  // ------------------------------------------
  // SyncMode : SERVER_TO_CLIENT 
  // ------------------------------------------
  12 : // Conflict triggerd by PLC ?  
       IF ( NOT AxesGroup.State.SyncStatePlc.InSync.Frame )
       THEN
         // search for changed index  
         FOR _rSyncIdx := 0 TO AxesGroup.State.UnifiedFrameIndex
         DO
           IF ( AxesGroup.State.DataChanged.Frame[_rSyncIdx] )
           THEN
             // set timeout
             SetTimeout(PT := _rTimeout, rTimer := _rTimer);
             // inc step counter
            _rStep := 20; // -> read RC data and write it to PLC                  
             EXIT;
					 END_IF
         END_FOR

         // Create log entry
         CreateLogMessagePara3 ( Timestamp   := SystemTime,
                                 MessageType := MessageType.CMD,
                                 Severity    := Severity.DEBUG,
                                 MessageCode := 0,
                                 MessageText := 'SyncFrameData: Synchronization of Frame[{1}] triggered by PLC, SyncMode = {2}, SyncTime = {3}, SyncDirection = RC -> PLC',
                                 Para1       :=  DINT_TO_STRING(_rSyncIdx),
                                 Para2       :=  SYNC_MODE_TO_STRING(AxesGroup.Parameter.Plc.Parameter.SynchronizationModes.Frame[SyncTime.AFTER_START_UP]),
                                 Para3       :=  SYNC_TIME_TO_STRING(SyncTime.AFTER_START_UP));
                                 RETURN;
       END_IF
   
       // Conflict triggered by RC ?
       IF ( NOT AxesGroup.State.SyncStateRc.InSync.Frame )
       THEN
         // get changed index 
        _rSyncIdx := LIMIT(0, AxesGroup.State.SyncStateRc.UnSyncNo.Frame, AxesGroup.State.UnifiedFrameIndex);
         // set timeout
         SetTimeout(PT := _rTimeout, rTimer := _rTimer);
         // inc step counter
        _rStep := 20; // -> read RC data and write it to PLC

         // Create log entry
         CreateLogMessagePara3 ( Timestamp   := SystemTime,
                                 MessageType := MessageType.CMD,
                                 Severity    := Severity.DEBUG,
                                 MessageCode := 0,
                                 MessageText := 'SyncFrameData: Synchronization of Frame[{1}] triggered by RC, SyncMode = {2}, SyncTime = {3}, SyncDirection = RC -> PLC',
                                 Para1       :=  DINT_TO_STRING(_rSyncIdx),
                                 Para2       :=  SYNC_MODE_TO_STRING(AxesGroup.Parameter.Plc.Parameter.SynchronizationModes.Frame[SyncTime.AFTER_START_UP]),
                                 Para3       :=  SYNC_TIME_TO_STRING(SyncTime.AFTER_START_UP));
                                 RETURN;
			 END_IF
       
       // set timeout
       SetTimeout(PT := _rTimeout, rTimer := _rTimer);
       // jump back
      _rStep := 10;
  

  // ------------------------------------------
  // SyncMode : AUTOMATIC 
  // ------------------------------------------
  13 : // Conflict triggerd by PLC ?  
       IF ( NOT AxesGroup.State.SyncStatePlc.InSync.Frame )
       THEN
         // search for changed index  
         FOR _rSyncIdx := 0 TO AxesGroup.State.UnifiedFrameIndex
         DO
           IF ( AxesGroup.State.DataChanged.Frame[_rSyncIdx] )
           THEN
             // set timeout
             SetTimeout(PT := _rTimeout, rTimer := _rTimer);
             // inc step counter
            _rStep := 30; // -> write PLC data to RC                  
             EXIT;
					 END_IF
         END_FOR
         
         // Create log entry
         CreateLogMessagePara3 ( Timestamp   := SystemTime,
                                 MessageType := MessageType.CMD,
                                 Severity    := Severity.DEBUG,
                                 MessageCode := 0,
                                 MessageText := 'SyncFrameData: Synchronization of Frame[{1}] triggered by PLC, SyncMode = {2}, SyncTime = {3}, SyncDirection = PLC -> RC',
                                 Para1       :=  DINT_TO_STRING(_rSyncIdx),
                                 Para2       :=  SYNC_MODE_TO_STRING(AxesGroup.Parameter.Plc.Parameter.SynchronizationModes.Frame[SyncTime.AFTER_START_UP]),
                                 Para3       :=  SYNC_TIME_TO_STRING(SyncTime.AFTER_START_UP));
                                 RETURN;
       END_IF
   
       // Conflict triggered by RC ?
       IF ( NOT AxesGroup.State.SyncStateRc.InSync.Frame )
       THEN
         // get changed index 
        _rSyncIdx := LIMIT(0, AxesGroup.State.SyncStateRc.UnSyncNo.Frame, AxesGroup.State.UnifiedFrameIndex);
         // set timeout
         SetTimeout(PT := _rTimeout, rTimer := _rTimer);
         // inc step counter
        _rStep := 20; // -> read RC data an write it to PLC

         // Create log entry
         CreateLogMessagePara3 ( Timestamp   := SystemTime,
                                 MessageType := MessageType.CMD,
                                 Severity    := Severity.DEBUG,
                                 MessageCode := 0,
                                 MessageText := 'SyncFrameData: Synchronization of Frame[{1}] triggered by RC, SyncMode = {2}, SyncTime = {3}, SyncDirection = RC -> PLC',
                                 Para1       :=  DINT_TO_STRING(_rSyncIdx),
                                 Para2       :=  SYNC_MODE_TO_STRING(AxesGroup.Parameter.Plc.Parameter.SynchronizationModes.Frame[SyncTime.AFTER_START_UP]),
                                 Para3       :=  SYNC_TIME_TO_STRING(SyncTime.AFTER_START_UP));
                                 RETURN;
			 END_IF
       
       // set timeout
       SetTimeout(PT := _rTimeout, rTimer := _rTimer);
       // jump back
      //_rStep := 10;


  // ------------------------------------------
  // Read Data from RC and write it to PLC
  // ------------------------------------------
  20 : IF (( NOT _readFrameData.Busy  ) AND 
           ( NOT _readFrameData.Error ))
       THEN
         // set command parameter
        _readFrameData.ParCmd.FrameNo := _rSyncIdx;      
         // execute command
        _readFrameData.Execute := TRUE;
         // set timeout
         SetTimeout(PT := _rTimeout, rTimer := _rTimer);
         // inc step counter
        _rStep := _rStep + 1;
       ELSE
         // check error ? 
         IF (_readFrameData.Error)
         THEN
           ErrorID     := _readFrameData.ErrorID;
           ErrorAddTxt := _readFrameData.ErrorAddTxt;
         END_IF  
       
         // timeout exceeded ? 
         IF (CheckTimeout(_rTimer) = RobotLibraryConstants.OK)
         THEN
           ErrorAddTxt := CONCAT(_stepName, DINT_TO_STRING(_rStep));
           SetError( ErrorID := RobotLibraryErrorIdEnum.ERR_TIMEOUT_CMD, Overwrite := FALSE);
         END_IF
       END_IF
 
  21 : IF (( NOT _readFrameData.Busy  ) AND
           ( NOT _readFrameData.Error ) AND
           (     _readFrameData.Done  ))
       THEN
         // reset execution
        _readFrameData.Execute := FALSE;
         // update internal frame data
         FrameData[_rSyncIdx].Data := _readFrameData.OutCmd.FrameData;         
        _frameData[_rSyncIdx].Data := _readFrameData.OutCmd.FrameData;
         // set available bit
         FrameData[_rSyncIdx].Available := TRUE;
        _frameData[_rSyncIdx].Available := TRUE;
         // set timeout
         SetTimeout(PT := _rTimeout, rTimer := _rTimer);
         // inc step counter
        _rStep := 10; // -> jump to after startup           
       ELSE
         // check error ? 
         IF (_readFrameData.Error)
         THEN
           ErrorID     := _readFrameData.ErrorID;
           ErrorAddTxt := _readFrameData.ErrorAddTxt;           
           // reset available bit
           FrameData[_rSyncIdx].Available := FALSE;
          _frameData[_rSyncIdx].Available := FALSE;
         END_IF  
       
         // timeout exceeded ? 
         IF (CheckTimeout(_rTimer) = RobotLibraryConstants.OK)
         THEN
           ErrorAddTxt := CONCAT(_stepName, DINT_TO_STRING(_rStep));
           SetError( ErrorID := RobotLibraryErrorIdEnum.ERR_TIMEOUT_CMD, Overwrite := FALSE);
         END_IF
       END_IF


  // ------------------------------------------
  // Write data from PLC to RC
  // ------------------------------------------
  30 : IF (( NOT _writeFrameData.Busy  ) AND 
           ( NOT _writeFrameData.Error ))
       THEN
         // set command parameter
        _writeFrameData.ParCmd.FrameNo   := _rSyncIdx;      
        _writeFrameData.ParCmd.FrameData :=  FrameData[_rSyncIdx].Data;
         // execute command
        _writeFrameData.Execute := TRUE;
         // set timeout
         SetTimeout(PT := _rTimeout, rTimer := _rTimer);
         // inc step counter
        _rStep := _rStep + 1;
       ELSE
         // check error ? 
         IF (_writeFrameData.Error)
         THEN
           ErrorID     := _writeFrameData.ErrorID;
           ErrorAddTxt := _writeFrameData.ErrorAddTxt;;
         END_IF  
       
         // timeout exceeded ? 
         IF (CheckTimeout(_rTimer) = RobotLibraryConstants.OK)
         THEN
           ErrorAddTxt := CONCAT(_stepName, DINT_TO_STRING(_rStep));
           SetError( ErrorID := RobotLibraryErrorIdEnum.ERR_TIMEOUT_CMD, Overwrite := FALSE);
         END_IF
       END_IF
 
  31 : IF (( NOT _writeFrameData.Busy  ) AND
           ( NOT _writeFrameData.Error ) AND
           (     _writeFrameData.Done  ))
       THEN
         // execute command
        _writeFrameData.Execute := FALSE;      
         // update internal frame data
        _frameData[_rSyncIdx] := FrameData[_rSyncIdx]; 
         // set available bit
         FrameData[_rSyncIdx].Available := TRUE; 
        _frameData[_rSyncIdx].Available := TRUE;         
         // set timeout
         SetTimeout(PT := _rTimeout, rTimer := _rTimer);
         // inc step counter
        _rStep := 10; // -> jump to after startup;           
       ELSE
         // check error ? 
         IF (_writeFrameData.Error)
         THEN
           SetWarning( WarningID := RobotLibraryWarningIdEnum.WARN_FRAME_SYNC_FAILED_BY_ERROR_OF_READ_OR_WRITE_CMD, Overwrite := TRUE);    
           // reset available bit
           FrameData[_rSyncIdx].Available := FALSE;
          _frameData[_rSyncIdx].Available := FALSE;
         END_IF  
       
         // timeout exceeded ? 
         IF (CheckTimeout(_rTimer) = RobotLibraryConstants.OK)
         THEN
           ErrorAddTxt := CONCAT(_stepName, DINT_TO_STRING(_rStep));
           SetError( ErrorID := RobotLibraryErrorIdEnum.ERR_TIMEOUT_CMD, Overwrite := FALSE);
         END_IF
       END_IF
       
ELSE
  // invalid step
  ErrorID     := RobotLibraryErrorIdEnum.ERR_INVALID_STEP;
  ErrorAddTxt := CONCAT(_stepName , DINT_TO_STRING(_stepCmd));
END_CASE  
                
END_METHOD

METHOD PRIVATE HandleSyncLoadData
VAR_IN_OUT
   /// Robot assignment of function
  AxesGroup : AxesGroup;
  /// LoadData stored on PLC.For more information refer to 5.5.6.4
  LoadData  : ARRAY[*] OF Load;
END_VAR 

VAR
  /// Internal step counter name
 _stepName        : STRING;    
  /// Internal reference to step counter
 _rStep           : REFERENCE TO DINT;
  /// Internal reference to timer
 _rTimer          : REFERENCE TO TON;
  /// Internal reference to timeout
 _rTimeout        : REFERENCE TO TIME; 
  /// Internal reference to synchroniztion index
 _rSyncIdx        : REFERENCE TO USINT;
  /// internal bit for condition found
 _found           : BOOL;
  /// empty data set to reset all DataChanged bits
 _dataChangedNone : AxesGroupStateDataChanged;
  /// internal index for loops
 _idx             : DINT;
  /// internal Start index for loops
 _idxStart        : USINT;
END_VAR
                  // Set internal references 
_stepName      :=   '_stepSyncLoadData = ';
_rStep       REF=    _stepSyncLoadData;
_rTimer      REF=   _timerSyncLoadData;
_rTimeout    REF= _timeoutSyncLoadData;
_rSyncIdx    REF=     _syncIdxLoadData;

CASE _rStep
OF    
  0: // Check initialisation configured ?
     IF (( _parCfg.PLC.Parameter.SynchronizationModes.Load[SyncTime.DURING_START_UP] = SyncMode.NO_SYNCHRONIZATION ) AND
         ( _parCfg.PLC.Parameter.SynchronizationModes.Load[SyncTime. AFTER_START_UP] = SyncMode.NO_SYNCHRONIZATION ))
     THEN
       RETURN;
     END_IF
     
     // Check More Data on RC than on PLC -> Synchronization not possible
     IF (AxesGroup.State.ConfigurationData.HighestToolIndex > AxesGroup.SystemData.LoadDataCount)
     THEN
       SetError( ErrorID := RobotLibraryErrorIdEnum.ERR_SYNC_LOAD_COUNT_RC_HIGHER_THAN_PLC, Overwrite := FALSE);
       RETURN;
		 END_IF

     // wait for initialisation done
     IF  ((     AxesGroup.State.RobotData.RCSupportedFunctions. ReadLoadData ) AND
          (     AxesGroup.State.RobotData.RCSupportedFunctions.WriteLoadData ) AND
          (     AxesGroup.State.Initialized                                  ) AND 
          ( NOT Error                                                        ))  
     THEN
       // Check PLC loads < RC Loads and SyncLoad enabled ?    
       IF (( AxesGroup.State.DataEnableSync.EnableSyncLoad      = TRUE                             )  AND
           ( AxesGroup.Parameter.Rob.Parameter.HighestLoadIndex > AxesGroup.SystemData.LoadDataMax ))        
       THEN
         SetWarning( WarningID := RobotLibraryWarningIdEnum.WARN_LOAD_DATA_ARRAY_TOO_SHORT, Overwrite := TRUE);
       END_IF

       // Create log entry
       CreateLogMessagePara1 ( Timestamp   := SystemTime,
                               MessageType := MessageType.CMD,
                               Severity    := Severity.DEBUG,
                               MessageCode := 0,
                               MessageText := 'SyncLoadData: Start initial reading of LoadData from RC',
                               Para1       :=  '');
                               
       //  calculate start index !!! Attention : 0 is not allowed - LoadData starts with 1 !!!
      _rSyncIdx := LIMIT(1 , DINT_TO_USINT(AxesGroup.SystemData.LoadDataMin), AxesGroup.State.UnifiedLoadIndex);
       // init count of unsynchronized elements
       AxesGroup.State.SyncStatePlc.UnSyncNo.Load := 0;
       // set timeout
       SetTimeout(PT := _rTimeout, rTimer := _rTimer);
       // inc step counter
      _rStep := _rStep + 1;
     END_IF     

     
     // Start read LoadData
  1: IF (( NOT _readLoadData.Busy  ) AND 
         ( NOT _readLoadData.Error ) AND
         ( NOT _readLoadData.Done  ))
     THEN
       // set command parameter
      _readLoadData.ParCmd.LoadNo := _rSyncIdx;      
       // execute command
      _readLoadData.Execute := TRUE;
       // set timeout
       SetTimeout(PT := _rTimeout, rTimer := _rTimer);
       // inc step counter
      _rStep := _rStep + 1;
     ELSE
       // check error ? 
       IF ( _readLoadData.Error )
       THEN
         SetWarning( WarningID := RobotLibraryWarningIdEnum.WARN_LOAD_SYNC_FAILED_BY_ERROR_OF_READ_OR_WRITE_CMD, Overwrite := FALSE );           
       END_IF  
       
       // timeout exceeded ? 
       IF (CheckTimeout(_rTimer) = RobotLibraryConstants.OK)
       THEN
         ErrorID     := RobotLibraryErrorIdEnum.ERR_TIMEOUT_CMD;
         ErrorAddTxt := CONCAT(_stepName, DINT_TO_STRING(_rStep));
       END_IF
     END_IF
 
     
     // Wait Loaddata read
  2: IF (( NOT _readLoadData.Busy  ) AND
         ( NOT _readLoadData.Error ) AND
         (     _readLoadData.Done  ))
     THEN
       // reset execution
      _readLoadData.Execute := FALSE;
       // set available bit
      _loadData[_rSyncIdx].Available := TRUE; 
       LoadData[_rSyncIdx].Available := TRUE;      
       // Copy data
      _loadData[_rSyncIdx].Data := _readLoadData.OutCmd.LoadData;

       // Check Load data is equal ? 
       IF ( NOT IsLoadDataEqual( Data1 := _loadData[_rSyncIdx].Data, Data2 := LoadData[_rSyncIdx].Data, IgnoreTimestamp := TRUE))
       THEN
         // Reset plc in sync flag
         AxesGroup.State.SyncStatePlc.InSync.Load := FALSE;
         // Set data changed flag
         AxesGroup.State.DataChanged.Load[_rSyncIdx] := TRUE;
         // inc count of unsynchronised plc Loads
         AxesGroup.State.SyncStatePlc.UnSyncNo.Load := AxesGroup.State.SyncStatePlc.UnSyncNo.Load + 1;
        
         // Create log entry
         CreateLogMessagePara1 ( Timestamp   := SystemTime,
                                 MessageType := MessageType.CMD,
                                 Severity    := Severity.DEBUG,
                                 MessageCode := 0,
                                 MessageText := 'SyncLoadData: Detected a difference in Load[{1}] between PLC and RC',
                                 Para1       :=  DINT_TO_STRING(_rSyncIdx));
        
        
         // Check synchronisation is enabled ? 
         IF ( NOT AxesGroup.State.DataEnableSync.EnableSyncLoad )
         THEN
           SetInfo( InfoID := RobotLibraryInfoIdEnum.INFO_SYNC_LOAD_DATA_DISABLED, Overwrite := FALSE);
				 END_IF
         
         // Check user interaction needed ?  
         IF ( AxesGroup.Parameter.PLC.Parameter.SyncUserInteraction.Load )
         THEN
           SetWarning( WarningID := RobotLibraryWarningIdEnum.WARN_LOAD_NUMBER_SYNC_ERROR, Overwrite := FALSE);                    
				 END_IF
			 END_IF
             
       // Check all Loads read ? 
       IF ( _rSyncIdx < AxesGroup.State.UnifiedLoadIndex )
       THEN
         // set timeout
         SetTimeout(PT := _rTimeout, rTimer := _rTimer);
         // inc Load index
        _rSyncIdx := _rSyncIdx + 1;
         // dec step counter
        _rStep := _rStep - 1;
       ELSE
         // set timeout
         SetTimeout(PT := _rTimeout, rTimer := _rTimer);
         // inc step counter
        _rStep := _rStep + 1;           
       END_IF
     ELSE
       // check error ? 
       IF (_readLoadData.Error)
       THEN
         // Set warning
         SetWarning( WarningID := RobotLibraryWarningIdEnum.WARN_LOAD_SYNC_FAILED_BY_ERROR_OF_READ_OR_WRITE_CMD, Overwrite := TRUE);                    
         // reset available bit
         LoadData[_rSyncIdx].Available := FALSE;
        _loadData[_rSyncIdx].Available := FALSE;
       END_IF  
       
       // timeout exceeded ? 
       IF (CheckTimeout(_rTimer) = RobotLibraryConstants.OK)
       THEN
         ErrorID     := RobotLibraryErrorIdEnum.ERR_TIMEOUT_CMD;
         ErrorAddTxt := CONCAT(_stepName, DINT_TO_STRING(_rStep));
       END_IF
     END_IF
     
     
     // Check synchronisation state ? 
  3: IF (( AxesGroup.State.SyncStatePlc.UnSyncNo.Load                                            = 0                           ) OR 
         ( AxesGroup.Parameter.Plc.Parameter.SynchronizationModes.Load[SyncTime.DURING_START_UP] = SyncMode.NO_SYNCHRONIZATION ))
     THEN
       // Update bit for data in sync
       AxesGroup.State.SyncStatePlc.InSync.Load := (AxesGroup.State.SyncStatePlc.UnSyncNo.Load = 0);
       // set timeout
       SetTimeout(PT := _rTimeout, rTimer := _rTimer);
       // inc step counter
      _rStep := 10; // -> jump to after startup
            
       // Create log entry
       CreateLogMessagePara1 ( Timestamp   := SystemTime,
                               MessageType := MessageType.CMD,
                               Severity    := Severity.DEBUG,
                               MessageCode := 0,
                               MessageText := 'SyncLoadData: Synchronization Startup Phase done',
                               Para1       :=  '' );      
     ELSE 
       // Check user interaction needed ? 
       IF ( NOT AxesGroup.Parameter.PLC.Parameter.SyncUserInteraction.Load )
       THEN
         CASE AxesGroup.Parameter.Plc.Parameter.SynchronizationModes.Load[SyncTime.DURING_START_UP] OF

           SyncMode.SERVER_TO_CLIENT : 

             // Overwrite PLC data with RC data
             FOR _idx := AxesGroup.SystemData.LoadDataMin TO AxesGroup.SystemData.LoadDataMax
             DO
               // Overwrite PLC data with RC data
               LoadData[_idx] := _loadData[_idx];            
						 END_FOR
        
             // Reset data changed flags
             AxesGroup.State.DataChanged.Load := _dataChangedNone.Load;
             // Reset Synchronizing flag
             AxesGroup.State.Synchronizing.Load := FALSE;
             // Set plc in sync flag
             AxesGroup.State.SyncStatePlc.InSync.Load := TRUE;
             // Reset count of unsynchronised plc Loads
             AxesGroup.State.SyncStatePlc.UnSyncNo.Load := 0;            
             // set timeout
             SetTimeout(PT := _rTimeout, rTimer := _rTimer);
             // inc step counter
            _rStep := 10; // -> jump to after startup         

            // Create log entry
            CreateLogMessagePara3 ( Timestamp   := SystemTime,
                                    MessageType := MessageType.CMD,
                                    Severity    := Severity.DEBUG,
                                    MessageCode := 0,
                                    MessageText := 'SyncLoadData: Synchronization of Loads triggered by StartUp-Compare, SyncMode = {2}, SyncTime = {3}, SyncDirection = RC -> PLC',
                                    Para1       :=  DINT_TO_STRING(_rSyncIdx),
                                    Para2       :=  SYNC_MODE_TO_STRING(AxesGroup.Parameter.Plc.Parameter.SynchronizationModes.Load[SyncTime.DURING_START_UP]),
                                    Para3       :=  SYNC_TIME_TO_STRING(SyncTime.DURING_START_UP));
            // Create log entry
            CreateLogMessagePara1 ( Timestamp   := SystemTime,
                                    MessageType := MessageType.CMD,
                                    Severity    := Severity.DEBUG,
                                    MessageCode := 0,
                                    MessageText := 'SyncLoadData: Applied the initial read Load data from RC',
                                    Para1       :=  '' );

				   SyncMode.CLIENT_TO_SERVER : ;

             //  calculate start index 
            _idxStart := LIMIT(1 , DINT_TO_USINT(AxesGroup.SystemData.LoadDataMin), AxesGroup.State.UnifiedLoadIndex);
      
             // Check conflicts to solve ? 
             FOR _rSyncIdx := _idxStart TO AxesGroup.State.UnifiedLoadIndex  // !!! Attention : 0 is not allowed - LoadData starts with 1 !!!
             DO
               IF ( AxesGroup.State.DataChanged.Load[_rSyncIdx] )
               THEN
                _found := TRUE;
                 EXIT;
		  			   END_IF
             END_FOR
           
             IF ( _found ) 
             THEN
               // Reset plc in sync flag
               AxesGroup.State.SyncStatePlc.InSync.Load := FALSE;
               // Set Synchronizing flag
               AxesGroup.State.Synchronizing.Load := TRUE;
               // set timeout
               SetTimeout(PT := _rTimeout, rTimer := _rTimer);
               // inc step counter
              _rStep := _rStep +1; // -> write PLC data to RC                  
               // Create log entry
               CreateLogMessagePara3 ( Timestamp   := SystemTime,
                                       MessageType := MessageType.CMD,
                                       Severity    := Severity.DEBUG,
                                       MessageCode := 0,
                                       MessageText := 'SyncLoadData: Synchronization of Load[{1}] triggered by StartUp-Compare, SyncMode = {2}, SyncTime = {3}, SyncDirection = PLC -> RC',
                                       Para1       :=  DINT_TO_STRING(_rSyncIdx),
                                       Para2       :=  SYNC_MODE_TO_STRING(AxesGroup.Parameter.Plc.Parameter.SynchronizationModes.Load[SyncTime.DURING_START_UP]),
                                       Para3       :=  SYNC_TIME_TO_STRING(SyncTime.DURING_START_UP));
             ELSE
               // Reset data changed flags
               AxesGroup.State.DataChanged.Load := _dataChangedNone.Load;
               // Reset Synchronizing flag
               AxesGroup.State.Synchronizing.Load := FALSE;
               // Set plc in sync flag
               AxesGroup.State.SyncStatePlc.InSync.Load := TRUE;
               // Reset count of unsynchronised Loads
               AxesGroup.State.SyncStatePlc.UnSyncNo.Load := 0;
               // set timeout
               SetTimeout(PT := _rTimeout, rTimer := _rTimer);
               // inc step counter
              _rStep := 10; // -> jump to after startup                  
				     END_IF
         ELSE
           // invalid sync mode for startup
           SetError( ErrorID := RobotLibraryErrorIdEnum.ERR_SYNC_MODE_INVALID, Overwrite := TRUE );
 	       END_CASE
       END_IF
     END_IF  

     
     // Start write Load data  
  4: IF (( NOT _writeLoadData.Busy  ) AND 
         ( NOT _writeLoadData.Error ))
     THEN
       // set command parameter
      _writeLoadData.ParCmd.LoadNo   := _rSyncIdx;      
      _writeLoadData.ParCmd.LoadData :=  LoadData[_rSyncIdx].Data;
       // execute command
      _writeLoadData.Execute := TRUE;
       // set timeout
       SetTimeout(PT := _rTimeout, rTimer := _rTimer);
       // inc step counter
      _rStep := _rStep + 1;
     ELSE
       // check error ? 
       IF (_writeLoadData.Error)
       THEN
         ErrorID     := _writeLoadData.ErrorID;
         ErrorAddTxt := _writeLoadData.ErrorAddTxt;;
       END_IF  
       
       // timeout exceeded ? 
       IF (CheckTimeout(_rTimer) = RobotLibraryConstants.OK)
       THEN
         ErrorID     := RobotLibraryErrorIdEnum.ERR_TIMEOUT_CMD;
         ErrorAddTxt := CONCAT(_stepName, DINT_TO_STRING(_rStep));
       END_IF
     END_IF
 
     
     // Wait Load data written ?   
  5: IF (( NOT _writeLoadData.Busy  ) AND
         ( NOT _writeLoadData.Error ) AND
         (     _writeLoadData.Done  ))
     THEN
       // execute command
      _writeLoadData.Execute := FALSE;
       // apply Load data to internal Load data
      _loadData[_rSyncIdx] := LoadData[_rSyncIdx];
       // reset data changed bit 
       AxesGroup.State.DataChanged.Load[_rSyncIdx] := FALSE;
       // dec count of unsynchronised Loads
       AxesGroup.State.SyncStatePlc.UnSyncNo.Load := AxesGroup.State.SyncStatePlc.UnSyncNo.Load - 1;
       // set timeout        
       SetTimeout(PT := _rTimeout, rTimer := _rTimer);
       // dec step counter
      _rStep := _rStep - 2; 
     ELSE
       // check error ? 
       IF (_writeLoadData.Error)
       THEN
         SetWarning( WarningID := RobotLibraryWarningIdEnum.WARN_LOAD_SYNC_FAILED_BY_ERROR_OF_READ_OR_WRITE_CMD, Overwrite := TRUE);           
       END_IF  
       
       // timeout exceeded ? 
       IF (CheckTimeout(_rTimer) = RobotLibraryConstants.OK)
       THEN
         ErrorID     := RobotLibraryErrorIdEnum.ERR_TIMEOUT_CMD;
         ErrorAddTxt := CONCAT(_stepName, DINT_TO_STRING(_rStep));
       END_IF
     END_IF

     
  // --------------------------------------------
  // SyncMode after startup : 
  // --------------------------------------------
         
  10 : // check synchronisation active ? 
       IF ( AxesGroup.Parameter.Plc.Parameter.SynchronizationModes.Load[SyncTime.AFTER_START_UP] = SyncMode.NO_SYNCHRONIZATION)
       THEN
         RETURN;
       END_IF
       
       // reset count of unsynchronised Loads
       AxesGroup.State.SyncStatePlc.UnSyncNo.Load := 0;

       //  calculate start index 
      _idxStart := LIMIT(1 , DINT_TO_USINT(AxesGroup.SystemData.LoadDataMin), AxesGroup.State.UnifiedLoadIndex);
       
       // Check all Load datas
       FOR _rSyncIdx := _idxStart TO AxesGroup.State.UnifiedLoadIndex // !!! Attention : 0 is not allowed - LoadData starts with 1 !!!  
       DO
         // compare Load data
         AxesGroup.State.DataChanged.Load[_rSyncIdx] := NOT IsLoadDataEqual( Data1 := LoadData[_rSyncIdx].Data, Data2 := _loadData[_rSyncIdx].Data, IgnoreTimestamp := FALSE);

         // Check Load data changed ? 
         IF (AxesGroup.State.DataChanged.Load[_rSyncIdx])
         THEN
           // inc count of unsynchronised plc Loads
           AxesGroup.State.SyncStatePlc.UnSyncNo.Load := AxesGroup.State.SyncStatePlc.UnSyncNo.Load + 1;
           // Create log entry
           CreateLogMessagePara2 ( Timestamp   := SystemTime,
                                   MessageType := MessageType.CMD,
                                   Severity    := Severity.DEBUG,
                                   MessageCode := 0,
                                   MessageText := 'SyncLoadData: Detected a local change of Load[{1}] on PLC, SyncTime = {2}',
                                   Para1       :=  DINT_TO_STRING(_rSyncIdx),    
                                   Para2       :=  SYNC_TIME_TO_STRING(SyncTime.AFTER_START_UP));       
				 END_IF

         // Update plc in sync flag
         AxesGroup.State.SyncStatePlc.InSync.Load := (AxesGroup.State.SyncStatePlc.UnSyncNo.Load = 0); 
	     END_FOR

       // Check synchronization is needed ? 
       IF ( NOT AxesGroup.State.SyncStatePlc.InSync.Load ) XOR  
          ( NOT AxesGroup.State.SyncStateRc .InSync.Load )
       THEN
         CASE AxesGroup.Parameter.Plc.Parameter.SynchronizationModes.Load[SyncTime.AFTER_START_UP] 
         OF         
           // NO_SYNCHRONIZATION
           SyncMode.NO_SYNCHRONIZATION : ; // no further action 
           
           // CLIENT_TO_SERVER
           SyncMode.CLIENT_TO_SERVER :
             // set timeout
             SetTimeout(PT := _rTimeout, rTimer := _rTimer);
             // inc step counter
            _rStep := 11;
  
           // SERVER_TO_CLIENT
           SyncMode.SERVER_TO_CLIENT :
             // set timeout
             SetTimeout(PT := _rTimeout, rTimer := _rTimer);
             // inc step counter
            _rStep := 12;
  
           // AUTOMATIC
           SyncMode.AUTOMATIC : 
             // set timeout
             SetTimeout(PT := _rTimeout, rTimer := _rTimer);
             // inc step counter
            _rStep := 13;
         END_CASE
       ELSE
         // datas changeḍ on both sides ? -> Warning 
         IF (( NOT AxesGroup.State.SyncStatePlc.InSync.Load ) AND  
             ( NOT AxesGroup.State.SyncStateRc .InSync.Load ))
         THEN
           SetWarning( WarningID := RobotLibraryWarningIdEnum.WARN_LOAD_SYNC_BOTH_SIDES_CHANGED, Overwrite :=  TRUE);
         END_IF
       END_IF


  // ------------------------------------------
  // SyncMode : CLIENT_TO_SERVER 
  // ------------------------------------------  
  11 : // Conflict triggerd by PLC ?  
       IF ( NOT AxesGroup.State.SyncStatePlc.InSync.Load )
       THEN
         //  calculate start index 
        _idxStart := LIMIT(1 , DINT_TO_USINT(AxesGroup.SystemData.LoadDataMin), AxesGroup.State.UnifiedLoadIndex);
       
         // search for changed index  
         FOR _rSyncIdx := _idxStart TO AxesGroup.State.UnifiedLoadIndex // !!! Attention : 0 is not allowed - LoadData starts with 1 !!!  
         DO
           IF ( AxesGroup.State.DataChanged.Load[_rSyncIdx] )
           THEN
             // set timeout
             SetTimeout(PT := _rTimeout, rTimer := _rTimer);
             // inc step counter
            _rStep := 30; // -> write PLC data to RC                  
             EXIT;             
					 END_IF
         END_FOR
         
         // Create log entry
         CreateLogMessagePara3 ( Timestamp   := SystemTime,
                                 MessageType := MessageType.CMD,
                                 Severity    := Severity.DEBUG,
                                 MessageCode := 0,
                                 MessageText := 'SyncLoadData: Synchronization of Load[{1}] triggered by PLC, SyncMode = {2}, SyncTime = {3}, SyncDirection = PLC -> RC',
                                 Para1       :=  DINT_TO_STRING(_rSyncIdx),
                                 Para2       :=  SYNC_MODE_TO_STRING(AxesGroup.Parameter.Plc.Parameter.SynchronizationModes.Load[SyncTime.AFTER_START_UP]),
                                 Para3       :=  SYNC_TIME_TO_STRING(SyncTime.AFTER_START_UP));
                                 RETURN;
       END_IF
   
       // Conflict triggered by RC ?
       IF ( NOT AxesGroup.State.SyncStateRc.InSync.Load )
       THEN
         // get changed index 
        _rSyncIdx :=  LIMIT(1 , AxesGroup.State.SyncStateRc.UnSyncNo.Load, AxesGroup.State.UnifiedLoadIndex); //  !!! Attention : 0 is not allowed - LoadData starts with 1 !!!  
         // set timeout
         SetTimeout(PT := _rTimeout, rTimer := _rTimer);
         // inc step counter
        _rStep := 30; // -> write PLC data to RC

         // Create log entry
         CreateLogMessagePara3 ( Timestamp   := SystemTime,
                                 MessageType := MessageType.CMD,
                                 Severity    := Severity.DEBUG,
                                 MessageCode := 0,
                                 MessageText := 'SyncLoadData: Synchronization of Load[{1}] triggered by RC, SyncMode = {2}, SyncTime = {3}, SyncDirection = PLC -> RC',
                                 Para1       :=  DINT_TO_STRING(_rSyncIdx),
                                 Para2       :=  SYNC_MODE_TO_STRING(AxesGroup.Parameter.Plc.Parameter.SynchronizationModes.Load[SyncTime.AFTER_START_UP]),
                                 Para3       :=  SYNC_TIME_TO_STRING(SyncTime.AFTER_START_UP));
                                 RETURN;
			 END_IF
       
       // set timeout
       SetTimeout(PT := _rTimeout, rTimer := _rTimer);
       // jump back
      _rStep := 10;

       
  // ------------------------------------------
  // SyncMode : SERVER_TO_CLIENT 
  // ------------------------------------------
  12 : // Conflict triggerd by PLC ?  
       IF ( NOT AxesGroup.State.SyncStatePlc.InSync.Load )
       THEN

         //  calculate start index 
        _idxStart := LIMIT(1 , DINT_TO_USINT(AxesGroup.SystemData.LoadDataMin), AxesGroup.State.UnifiedLoadIndex);
       
         // search for changed index  
         FOR _rSyncIdx := _idxStart TO AxesGroup.State.UnifiedLoadIndex // !!! Attention : 0 is not allowed - LoadData starts with 1 !!!  
         DO
           IF ( AxesGroup.State.DataChanged.Load[_rSyncIdx] )
           THEN
             // set timeout
             SetTimeout(PT := _rTimeout, rTimer := _rTimer);
             // inc step counter
            _rStep := 20; // -> read RC data and write it to PLC                  
             EXIT;
					 END_IF
         END_FOR

         // Create log entry
         CreateLogMessagePara3 ( Timestamp   := SystemTime,
                                 MessageType := MessageType.CMD,
                                 Severity    := Severity.DEBUG,
                                 MessageCode := 0,
                                 MessageText := 'SyncLoadData: Synchronization of Load[{1}] triggered by PLC, SyncMode = {2}, SyncTime = {3}, SyncDirection = RC -> PLC',
                                 Para1       :=  DINT_TO_STRING(_rSyncIdx),
                                 Para2       :=  SYNC_MODE_TO_STRING(AxesGroup.Parameter.Plc.Parameter.SynchronizationModes.Load[SyncTime.AFTER_START_UP]),
                                 Para3       :=  SYNC_TIME_TO_STRING(SyncTime.AFTER_START_UP));
                                 RETURN;
       END_IF
   
       // Conflict triggered by RC ?
       IF ( NOT AxesGroup.State.SyncStateRc.InSync.Load )
       THEN
         // get changed index 
        _rSyncIdx := LIMIT(1 , AxesGroup.State.SyncStateRc.UnSyncNo.Load, AxesGroup.State.UnifiedLoadIndex); //  !!! Attention : 0 is not allowed - LoadData starts with 1 !!!  
         // set timeout
         SetTimeout(PT := _rTimeout, rTimer := _rTimer);
         // inc step counter
        _rStep := 20; // -> read RC data and write it to PLC

         // Create log entry
         CreateLogMessagePara3 ( Timestamp   := SystemTime,
                                 MessageType := MessageType.CMD,
                                 Severity    := Severity.DEBUG,
                                 MessageCode := 0,
                                 MessageText := 'SyncLoadData: Synchronization of Load[{1}] triggered by RC, SyncMode = {2}, SyncTime = {3}, SyncDirection = RC -> PLC',
                                 Para1       :=  DINT_TO_STRING(_rSyncIdx),
                                 Para2       :=  SYNC_MODE_TO_STRING(AxesGroup.Parameter.Plc.Parameter.SynchronizationModes.Load[SyncTime.AFTER_START_UP]),
                                 Para3       :=  SYNC_TIME_TO_STRING(SyncTime.AFTER_START_UP));
                                 RETURN;
			 END_IF
       
       // set timeout
       SetTimeout(PT := _rTimeout, rTimer := _rTimer);
       // jump back
      _rStep := 10;
  

  // ------------------------------------------
  // SyncMode : AUTOMATIC 
  // ------------------------------------------
  13 : // Conflict triggerd by PLC ?  
       IF ( NOT AxesGroup.State.SyncStatePlc.InSync.Load )
       THEN
       
         //  calculate start index 
        _idxStart := LIMIT(1 , DINT_TO_USINT(AxesGroup.SystemData.LoadDataMin), AxesGroup.State.UnifiedLoadIndex);

         // search for changed index  
         FOR _rSyncIdx := _idxStart TO AxesGroup.State.UnifiedLoadIndex // !!! Attention : 0 is not allowed - LoadData starts with 1 !!!  
         DO
           IF ( AxesGroup.State.DataChanged.Load[_rSyncIdx] )
           THEN
             // set timeout
             SetTimeout(PT := _rTimeout, rTimer := _rTimer);
             // inc step counter
            _rStep := 30; // -> write PLC data to RC                  
             EXIT;
					 END_IF
         END_FOR
         
         // Create log entry
         CreateLogMessagePara3 ( Timestamp   := SystemTime,
                                 MessageType := MessageType.CMD,
                                 Severity    := Severity.DEBUG,
                                 MessageCode := 0,
                                 MessageText := 'SyncLoadData: Synchronization of Load[{1}] triggered by PLC, SyncMode = {2}, SyncTime = {3}, SyncDirection = PLC -> RC',
                                 Para1       :=  DINT_TO_STRING(_rSyncIdx),
                                 Para2       :=  SYNC_MODE_TO_STRING(AxesGroup.Parameter.Plc.Parameter.SynchronizationModes.Load[SyncTime.AFTER_START_UP]),
                                 Para3       :=  SYNC_TIME_TO_STRING(SyncTime.AFTER_START_UP));
                                 RETURN;
       END_IF
   
       // Conflict triggered by RC ?
       IF ( NOT AxesGroup.State.SyncStateRc.InSync.Load )
       THEN
         // get changed index 
        _rSyncIdx := LIMIT(1 , AxesGroup.State.SyncStateRc.UnSyncNo.Load, AxesGroup.State.UnifiedLoadIndex); //  !!! Attention : 0 is not allowed - LoadData starts with 1 !!!  
         // set timeout
         SetTimeout(PT := _rTimeout, rTimer := _rTimer);
         // inc step counter
        _rStep := 20; // -> read RC data an write it to PLC

         // Create log entry
         CreateLogMessagePara3 ( Timestamp   := SystemTime,
                                 MessageType := MessageType.CMD,
                                 Severity    := Severity.DEBUG,
                                 MessageCode := 0,
                                 MessageText := 'SyncLoadData: Synchronization of Load[{1}] triggered by RC, SyncMode = {2}, SyncTime = {3}, SyncDirection = RC -> PLC',
                                 Para1       :=  DINT_TO_STRING(_rSyncIdx),
                                 Para2       :=  SYNC_MODE_TO_STRING(AxesGroup.Parameter.Plc.Parameter.SynchronizationModes.Load[SyncTime.AFTER_START_UP]),
                                 Para3       :=  SYNC_TIME_TO_STRING(SyncTime.AFTER_START_UP));
                                 RETURN;
			 END_IF
       
       // set timeout
       SetTimeout(PT := _rTimeout, rTimer := _rTimer);
       // jump back
      //_rStep := 10;


  // ------------------------------------------
  // Read Data from RC and write it to PLC
  // ------------------------------------------
  20 : IF (( NOT _readLoadData.Busy  ) AND 
           ( NOT _readLoadData.Error ))
       THEN
         // set command parameter
        _readLoadData.ParCmd.LoadNo := _rSyncIdx;      
         // execute command
        _readLoadData.Execute := TRUE;
         // set timeout
         SetTimeout(PT := _rTimeout, rTimer := _rTimer);
         // inc step counter
        _rStep := _rStep + 1;
       ELSE
         // check error ? 
         IF (_readLoadData.Error)
         THEN
           ErrorID     := _readLoadData.ErrorID;
           ErrorAddTxt := _readLoadData.ErrorAddTxt;
         END_IF  
       
         // timeout exceeded ? 
         IF (CheckTimeout(_rTimer) = RobotLibraryConstants.OK)
         THEN
           ErrorID     := RobotLibraryErrorIdEnum.ERR_TIMEOUT_CMD;
           ErrorAddTxt := CONCAT(_stepName, DINT_TO_STRING(_rStep));
         END_IF
       END_IF
 
  21 : IF (( NOT _readLoadData.Busy  ) AND
           ( NOT _readLoadData.Error ) AND
           (     _readLoadData.Done  ))
       THEN
         // reset execution
        _readLoadData.Execute := FALSE;
         // update internal Load data
         LoadData[_rSyncIdx].Data := _readLoadData.OutCmd.LoadData;         
        _loadData[_rSyncIdx].Data := _readLoadData.OutCmd.LoadData;
         // set available bit
         LoadData[_rSyncIdx].Available := TRUE;
        _loadData[_rSyncIdx].Available := TRUE;
         // set timeout
         SetTimeout(PT := _rTimeout, rTimer := _rTimer);
         // inc step counter
        _rStep := 10; // -> jump to after startup           
       ELSE
         // check error ? 
         IF (_readLoadData.Error)
         THEN
           ErrorID     := _readLoadData.ErrorID;
           ErrorAddTxt := _readLoadData.ErrorAddTxt;           
           // reset available bit
           LoadData[_rSyncIdx].Available := FALSE;
          _loadData[_rSyncIdx].Available := FALSE;
         END_IF  
       
         // timeout exceeded ? 
         IF (CheckTimeout(_rTimer) = RobotLibraryConstants.OK)
         THEN
           ErrorID     := RobotLibraryErrorIdEnum.ERR_TIMEOUT_CMD;
           ErrorAddTxt := CONCAT(_stepName, DINT_TO_STRING(_rStep));
         END_IF
       END_IF


  // ------------------------------------------
  // Write data from PLC to RC
  // ------------------------------------------
  30 : IF (( NOT _writeLoadData.Busy  ) AND 
           ( NOT _writeLoadData.Error ))
       THEN
         // set command parameter
        _writeLoadData.ParCmd.LoadNo   := _rSyncIdx;      
        _writeLoadData.ParCmd.LoadData :=  LoadData[_rSyncIdx].Data;
         // execute command
        _writeLoadData.Execute := TRUE;
         // set timeout
         SetTimeout(PT := _rTimeout, rTimer := _rTimer);
         // inc step counter
        _rStep := _rStep + 1;
       ELSE
         // check error ? 
         IF (_writeLoadData.Error)
         THEN
           ErrorID     := _writeLoadData.ErrorID;
           ErrorAddTxt := _writeLoadData.ErrorAddTxt;;
         END_IF  
       
         // timeout exceeded ? 
         IF (CheckTimeout(_rTimer) = RobotLibraryConstants.OK)
         THEN
           ErrorID     := RobotLibraryErrorIdEnum.ERR_TIMEOUT_CMD;
           ErrorAddTxt := CONCAT(_stepName, DINT_TO_STRING(_rStep));
         END_IF
       END_IF
 
  31 : IF (( NOT _writeLoadData.Busy  ) AND
           ( NOT _writeLoadData.Error ) AND
           (     _writeLoadData.Done  ))
       THEN
         // execute command
        _writeLoadData.Execute := FALSE;      
         // update internal Load data
        _loadData[_rSyncIdx] := LoadData[_rSyncIdx]; 
         // set available bit
         LoadData[_rSyncIdx].Available := TRUE; 
        _loadData[_rSyncIdx].Available := TRUE;         
         // set timeout
         SetTimeout(PT := _rTimeout, rTimer := _rTimer);
         // inc step counter
        _rStep := 10; // -> jump to after startup;           
       ELSE
         // check error ? 
         IF (_writeLoadData.Error)
         THEN
           SetWarning( WarningID := RobotLibraryWarningIdEnum.WARN_LOAD_SYNC_FAILED_BY_ERROR_OF_READ_OR_WRITE_CMD, Overwrite := TRUE);    
           // reset available bit
           LoadData[_rSyncIdx].Available := FALSE;
          _loadData[_rSyncIdx].Available := FALSE;
         END_IF  
       
         // timeout exceeded ? 
         IF (CheckTimeout(_rTimer) = RobotLibraryConstants.OK)
         THEN
           ErrorID     := RobotLibraryErrorIdEnum.ERR_TIMEOUT_CMD;
           ErrorAddTxt := CONCAT(_stepName, DINT_TO_STRING(_rStep));
         END_IF
       END_IF
       
ELSE
  // invalid step
  ErrorID     := RobotLibraryErrorIdEnum.ERR_INVALID_STEP;
  ErrorAddTxt := CONCAT(_stepName , DINT_TO_STRING(_stepCmd));
END_CASE  
                
END_METHOD

METHOD PRIVATE HandleSyncRobotDefaultDynamics
VAR_IN_OUT
   /// Robot assignment of function
  AxesGroup       : AxesGroup;
  /// Default dynamics stored on PLC. For more information refer to 5.5.7
  DefaultDynamics : DefaultDynamics;
END_VAR 

VAR
  /// Internal step counter name
 _stepName        : STRING;    
  /// Internal reference to step counter
 _rStep           : REFERENCE TO DINT;
  /// Internal reference to timer
 _rTimer          : REFERENCE TO TON;
  /// Internal reference to timeout
 _rTimeout        : REFERENCE TO TIME; 
  /// Internal reference to synchroniztion index
 _rSyncIdx        : REFERENCE TO USINT;
  /// internal bit for condition found
 _found           : BOOL;
  /// empty data set to reset all DataChanged bits
 _dataChangedNone : AxesGroupStateDataChanged;
END_VAR
                  // Set internal references 
_stepName      :=   '_stepSyncDefaultDynamics = ';
_rStep       REF=    _stepSyncDefaultDynamics;
_rTimer      REF=   _timerSyncDefaultDynamics;
_rTimeout    REF= _timeoutSyncDefaultDynamics;

CASE _rStep
OF    
  0: // Check initialisation configured ?
     IF (( _parCfg.PLC.Parameter.SynchronizationModes.DefaultDynamics[SyncTime.DURING_START_UP] = SyncMode.NO_SYNCHRONIZATION ) AND
         ( _parCfg.PLC.Parameter.SynchronizationModes.DefaultDynamics[SyncTime. AFTER_START_UP] = SyncMode.NO_SYNCHRONIZATION ))
     THEN
       RETURN;
     END_IF

     // wait for initialisation done
     IF  ((     AxesGroup.State.RobotData.RCSupportedFunctions .ReadRobotDefaultDynamics ) AND
          (     AxesGroup.State.RobotData.RCSupportedFunctions.WriteRobotDefaultDynamics ) AND
          (     AxesGroup.State.Initialized                                              ) AND 
          ( NOT Error                                                                    ))  
     THEN
       // Create log entry
       CreateLogMessagePara1 ( Timestamp   := SystemTime,
                               MessageType := MessageType.CMD,
                               Severity    := Severity.DEBUG,
                               MessageCode := 0,
                               MessageText := 'SyncDefaultDynamics: Start initial reading of DefaultDynamics from RC',
                               Para1       :=  '');
       
       // set timeout
       SetTimeout(PT := _rTimeout, rTimer := _rTimer);
       // inc step counter
      _rStep := _rStep + 1;
     END_IF     

     
     // Start read DefaultDynamics
  1: IF (( NOT _readRobotDefaultDynamics.Busy  ) AND 
         ( NOT _readRobotDefaultDynamics.Error ) AND
         ( NOT _readRobotDefaultDynamics.Done  ))
     THEN
       // execute command
      _readRobotDefaultDynamics.Execute := TRUE;
       // set timeout
       SetTimeout(PT := _rTimeout, rTimer := _rTimer);
       // inc step counter
      _rStep := _rStep + 1;
     ELSE
       // check error ? 
       IF ( _readRobotDefaultDynamics.Error )
       THEN
         SetWarning( WarningID := RobotLibraryWarningIdEnum.WARN_DEFAULT_DYNAMICS_SYNC_FAILED_BY_ERROR_OF_READ_OR_WRITE_CMD, Overwrite := FALSE );           
       END_IF  
       
       // timeout exceeded ? 
       IF (CheckTimeout(_rTimer) = RobotLibraryConstants.OK)
       THEN
         ErrorID     := RobotLibraryErrorIdEnum.ERR_TIMEOUT_CMD;
         ErrorAddTxt := CONCAT(_stepName, DINT_TO_STRING(_rStep));
       END_IF
     END_IF
 
     
     // Wait DefaultDynamics read
  2: IF (( NOT _readRobotDefaultDynamics.Busy  ) AND
         ( NOT _readRobotDefaultDynamics.Error ) AND
         (     _readRobotDefaultDynamics.Done  ))
     THEN
       // reset execution
      _readRobotDefaultDynamics.Execute := FALSE;
       // Copy data
      _defaultDynamics := _readRobotDefaultDynamics.OutCmd.DynamicValues;
       // Set plc in sync flag
       AxesGroup.State.SyncStatePlc.InSync.DefaultDynamics := TRUE;
       // inc step counter
      _rStep := _rStep + 1;           

       // Check DefaultDynamics data is equal ? 
       IF ( NOT IsDefaultDynamicsEqual( Data1 := _defaultDynamics, Data2 := DefaultDynamics, IgnoreTimestamp := TRUE))
       THEN
         // Reset plc in sync flag
         AxesGroup.State.SyncStatePlc.InSync.DefaultDynamics := FALSE;
         // Set data changed flag
         AxesGroup.State.DataChanged.DefaultDynamics := TRUE;
         // set timeout
         SetTimeout(PT := _rTimeout, rTimer := _rTimer);
        
         // Create log entry
         CreateLogMessagePara1 ( Timestamp   := SystemTime,
                                 MessageType := MessageType.CMD,
                                 Severity    := Severity.DEBUG,
                                 MessageCode := 0,
                                 MessageText := 'SyncDefaultDynamics: Detected a difference in DefaultDynamics between PLC and RC',
                                 Para1       :=  '');
        
        
         // Check synchronisation is enabled ? 
         IF ( NOT  AxesGroup.State.DataEnableSync.EnableSyncDefaultDynamics )
         THEN
           SetInfo( InfoID := RobotLibraryInfoIdEnum.INFO_SYNC_DEFAULT_DYNAMICS_DISABLED, Overwrite := FALSE);
				 END_IF
         
         // Check user interaction needed ?  
         IF ( AxesGroup.Parameter.Plc.Parameter.SyncUserInteraction.DefaultDynamics )
         THEN
           SetWarning( WarningID := RobotLibraryWarningIdEnum.WARN_DEFAULT_DYNAMICS_SYNC_ERROR, Overwrite := FALSE);                    
				 END_IF
			 END_IF             
     ELSE
       // check error ? 
       IF (_readRobotDefaultDynamics.Error)
       THEN
         // Set warning
         SetWarning( WarningID := RobotLibraryWarningIdEnum.WARN_DEFAULT_DYNAMICS_SYNC_FAILED_BY_ERROR_OF_READ_OR_WRITE_CMD, Overwrite := TRUE);                    
       END_IF  
       
       // timeout exceeded ? 
       IF (CheckTimeout(_rTimer) = RobotLibraryConstants.OK)
       THEN
         ErrorID     := RobotLibraryErrorIdEnum.ERR_TIMEOUT_CMD;
         ErrorAddTxt := CONCAT(_stepName, DINT_TO_STRING(_rStep));
       END_IF
     END_IF
     
     
     // Check synchronisation state ? 
  3: IF ((  NOT AxesGroup.State.DataChanged.DefaultDynamics                                                                                    ) OR 
         (      AxesGroup.Parameter.Plc.Parameter.SynchronizationModes.DefaultDynamics[SyncTime.DURING_START_UP] = SyncMode.NO_SYNCHRONIZATION ))
     THEN
       // Update bit for data in sync
       AxesGroup.State.SyncStatePlc.InSync.DefaultDynamics := NOT AxesGroup.State.DataChanged.DefaultDynamics ;
       // set timeout
       SetTimeout(PT := _rTimeout, rTimer := _rTimer);
       // inc step counter
      _rStep := 10; // -> jump to after startup
            
       // Create log entry
       CreateLogMessagePara1 ( Timestamp   := SystemTime,
                               MessageType := MessageType.CMD,
                               Severity    := Severity.DEBUG,
                               MessageCode := 0,
                               MessageText := 'SyncDefaultDynamics: Synchronization Startup Phase done',
                               Para1       :=  '' );      
     ELSE 
       // Check user interaction needed ? 
       IF ( NOT AxesGroup.Parameter.Plc.Parameter.SyncUserInteraction.DefaultDynamics )
       THEN 
         CASE AxesGroup.Parameter.Plc.Parameter.SynchronizationModes.DefaultDynamics[SyncTime.DURING_START_UP] OF

           SyncMode.SERVER_TO_CLIENT : 

             // Overwrite PLC data with RC data
             DefaultDynamics := _defaultDynamics;            
             // Reset data changed flags
             AxesGroup.State.DataChanged.DefaultDynamics := _dataChangedNone.DefaultDynamics;
             // Reset Synchronizing flag
             AxesGroup.State.Synchronizing.DefaultDynamics := FALSE;
             // Set plc in sync flag
             AxesGroup.State.SyncStatePlc.InSync.DefaultDynamics := TRUE;
             // set timeout
             SetTimeout(PT := _rTimeout, rTimer := _rTimer);
             // inc step counter
            _rStep := 10; // -> jump to after startup         

            // Create log entry
            CreateLogMessagePara2 ( Timestamp   := SystemTime,
                                    MessageType := MessageType.CMD,
                                    Severity    := Severity.DEBUG,
                                    MessageCode := 0,
                                    MessageText := 'SyncDefaultDynamics: Synchronization of DefaultDynamics triggered by StartUp-Compare, SyncMode = {1}, SyncTime = {2}, SyncDirection = RC -> PLC',
                                    Para1       :=  SYNC_MODE_TO_STRING(AxesGroup.Parameter.Plc.Parameter.SynchronizationModes.DefaultDynamics[SyncTime.DURING_START_UP]),
                                    Para2       :=  SYNC_TIME_TO_STRING(SyncTime.DURING_START_UP));
            // Create log entry
            CreateLogMessagePara1 ( Timestamp   := SystemTime,
                                    MessageType := MessageType.CMD,
                                    Severity    := Severity.DEBUG,
                                    MessageCode := 0,
                                    MessageText := 'SyncDefaultDynamics: Applied the initial read DefaultDynamics from RC',
                                    Para1       :=  '' );

				   SyncMode.CLIENT_TO_SERVER : ;

             IF ( AxesGroup.State.DataChanged.DefaultDynamics ) 
             THEN
               // Reset plc in sync flag
               AxesGroup.State.SyncStatePlc.InSync.DefaultDynamics := FALSE;
               // Set Synchronizing flag
               AxesGroup.State.Synchronizing.DefaultDynamics := TRUE;
               // set timeout
               SetTimeout(PT := _rTimeout, rTimer := _rTimer);
               // inc step counter
              _rStep := _rStep +1; // -> write PLC data to RC                  
               // Create log entry
               CreateLogMessagePara2 ( Timestamp   := SystemTime,
                                       MessageType := MessageType.CMD,
                                       Severity    := Severity.DEBUG,
                                       MessageCode := 0,
                                       MessageText := 'SyncDefaultDynamics: Synchronization of DefaultDynamics triggered by StartUp-Compare, SyncMode = {1}, SyncTime = {2}, SyncDirection = PLC -> RC',
                                       Para1       :=  SYNC_MODE_TO_STRING(AxesGroup.Parameter.Plc.Parameter.SynchronizationModes.DefaultDynamics[SyncTime.DURING_START_UP]),
                                       Para2       :=  SYNC_TIME_TO_STRING(SyncTime.DURING_START_UP));
             ELSE
               // Reset data changed flags
               AxesGroup.State.DataChanged.DefaultDynamics := _dataChangedNone.DefaultDynamics;
               // Reset Synchronizing flag
               AxesGroup.State.Synchronizing.DefaultDynamics := FALSE;
               // Set plc in sync flag
               AxesGroup.State.SyncStatePlc.InSync.DefaultDynamics := TRUE;
               // set timeout
               SetTimeout(PT := _rTimeout, rTimer := _rTimer);
               // inc step counter
              _rStep := 10; // -> jump to after startup                  
				     END_IF
         ELSE
           // invalid sync mode for startup
           SetError( ErrorID := RobotLibraryErrorIdEnum.ERR_SYNC_MODE_INVALID, Overwrite := TRUE );
 	       END_CASE
       END_IF
     END_IF  

     
     // Start write DefaultDynamics data  
  4: IF (( NOT _writeRobotDefaultDynamics.Busy  ) AND 
         ( NOT _writeRobotDefaultDynamics.Error ))
     THEN
       // set command parameter
      _writeRobotDefaultDynamics.ParCmd.DynamicValues :=  DefaultDynamics;
       // execute command
      _writeRobotDefaultDynamics.Execute := TRUE;
       // set timeout
       SetTimeout(PT := _rTimeout, rTimer := _rTimer);
       // inc step counter
      _rStep := _rStep + 1;
     ELSE
       // check error ? 
       IF (_writeRobotDefaultDynamics.Error)
       THEN
         ErrorID     := _writeRobotDefaultDynamics.ErrorID;
         ErrorAddTxt := _writeRobotDefaultDynamics.ErrorAddTxt;;
       END_IF  
       
       // timeout exceeded ? 
       IF (CheckTimeout(_rTimer) = RobotLibraryConstants.OK)
       THEN
         ErrorID     := RobotLibraryErrorIdEnum.ERR_TIMEOUT_CMD;
         ErrorAddTxt := CONCAT(_stepName, DINT_TO_STRING(_rStep));
       END_IF
     END_IF
 
     
     // Wait DefaultDynamics data written ?   
  5: IF (( NOT _writeRobotDefaultDynamics.Busy  ) AND
         ( NOT _writeRobotDefaultDynamics.Error ) AND
         (     _writeRobotDefaultDynamics.Done  ))
     THEN
       // execute command
      _writeRobotDefaultDynamics.Execute := FALSE;
       // apply DefaultDynamics data to internal DefaultDynamics data
      _defaultDynamics := DefaultDynamics;
       // reset data changed bit 
       AxesGroup.State.DataChanged.DefaultDynamics := FALSE;
       // set timeout        
       SetTimeout(PT := _rTimeout, rTimer := _rTimer);
       // dec step counter
      _rStep := _rStep - 2; 
     ELSE
       // check error ? 
       IF (_writeRobotDefaultDynamics.Error)
       THEN
         SetWarning( WarningID := RobotLibraryWarningIdEnum.WARN_DEFAULT_DYNAMICS_SYNC_FAILED_BY_ERROR_OF_READ_OR_WRITE_CMD, Overwrite := TRUE);           
       END_IF  
       
       // timeout exceeded ? 
       IF (CheckTimeout(_rTimer) = RobotLibraryConstants.OK)
       THEN
         ErrorID     := RobotLibraryErrorIdEnum.ERR_TIMEOUT_CMD;
         ErrorAddTxt := CONCAT(_stepName, DINT_TO_STRING(_rStep));
       END_IF
     END_IF

     
  // --------------------------------------------
  // SyncMode after startup : 
  // --------------------------------------------
         
  10 :// check synchronisation active ? 
       IF ( AxesGroup.Parameter.Plc.Parameter.SynchronizationModes.DefaultDynamics[SyncTime.AFTER_START_UP] = SyncMode.NO_SYNCHRONIZATION)
       THEN
         RETURN;
       END_IF
       
       // compare DefaultDynamics data
       AxesGroup.State.DataChanged.DefaultDynamics := NOT IsDefaultDynamicsEqual( Data1 := DefaultDynamics, Data2 := _defaultDynamics, IgnoreTimestamp := FALSE);

       // Check DefaultDynamics data changed ? 
       IF (AxesGroup.State.DataChanged.DefaultDynamics)
       THEN
         // Create log entry
         CreateLogMessagePara1 ( Timestamp   := SystemTime,
                                 MessageType := MessageType.CMD,
                                 Severity    := Severity.DEBUG,
                                 MessageCode := 0,
                                 MessageText := 'SyncDefaultDynamics: Detected a local change of DefaultDynamics on PLC, SyncTime = {1}',
                                 Para1       :=  SYNC_TIME_TO_STRING(SyncTime.AFTER_START_UP));       
       END_IF

       // Update plc in sync flag
       AxesGroup.State.SyncStatePlc.InSync.DefaultDynamics := NOT AxesGroup.State.DataChanged.DefaultDynamics; 


       // Check synchronization is needed ? 
       IF ( NOT AxesGroup.State.SyncStatePlc.InSync.DefaultDynamics ) XOR  
          ( NOT AxesGroup.State.SyncStateRc .InSync.DefaultDynamics )
       THEN
         CASE AxesGroup.Parameter.Plc.Parameter.SynchronizationModes.DefaultDynamics[SyncTime.AFTER_START_UP] 
         OF         
           // NO_SYNCHRONIZATION
           SyncMode.NO_SYNCHRONIZATION : ; // no further action 
           
           // CLIENT_TO_SERVER
           SyncMode.CLIENT_TO_SERVER :
             // set timeout
             SetTimeout(PT := _rTimeout, rTimer := _rTimer);
             // inc step counter
            _rStep := 11;
  
           // SERVER_TO_CLIENT
           SyncMode.SERVER_TO_CLIENT :
             // set timeout
             SetTimeout(PT := _rTimeout, rTimer := _rTimer);
             // inc step counter
            _rStep := 12;
  
           // AUTOMATIC
           SyncMode.AUTOMATIC : 
             // set timeout
             SetTimeout(PT := _rTimeout, rTimer := _rTimer);
             // inc step counter
            _rStep := 13;
         END_CASE
       ELSE
         // datas changeḍ on both sides ? -> Warning 
         IF (( NOT AxesGroup.State.SyncStatePlc.InSync.DefaultDynamics ) AND  
             ( NOT AxesGroup.State.SyncStateRc .InSync.DefaultDynamics ))
         THEN
           SetWarning( WarningID := RobotLibraryWarningIdEnum.WARN_DEFAULT_DYNAMICS_SYNC_BOTH_SIDES_CHANGED, Overwrite := TRUE);
         END_IF
       END_IF


  // ------------------------------------------
  // SyncMode : CLIENT_TO_SERVER 
  // ------------------------------------------  
  11 : // Conflict triggerd by PLC ?  
       IF ( NOT AxesGroup.State.SyncStatePlc.InSync.DefaultDynamics ) 
       THEN
         // set timeout
         SetTimeout(PT := _rTimeout, rTimer := _rTimer);
         // inc step counter
        _rStep := 30; // -> write PLC data to RC                  
         
         // Create log entry
         CreateLogMessagePara2 ( Timestamp   := SystemTime,
                                 MessageType := MessageType.CMD,
                                 Severity    := Severity.DEBUG,
                                 MessageCode := 0,
                                 MessageText := 'SyncDefaultDynamics: Synchronization of DefaultDynamics triggered by PLC, SyncMode = {1}, SyncTime = {2}, SyncDirection = PLC -> RC',
                                 Para1       :=  SYNC_MODE_TO_STRING(AxesGroup.Parameter.Plc.Parameter.SynchronizationModes.DefaultDynamics[SyncTime.AFTER_START_UP]),
                                 Para2       :=  SYNC_TIME_TO_STRING(SyncTime.AFTER_START_UP));
                                 RETURN;
       END_IF
   
       // Conflict triggered by RC ?
       IF ( NOT AxesGroup.State.SyncStateRc.InSync.DefaultDynamics )
       THEN
         // set timeout
         SetTimeout(PT := _rTimeout, rTimer := _rTimer);
         // inc step counter
        _rStep := 30; // -> write PLC data to RC

         // Create log entry
         CreateLogMessagePara2 ( Timestamp   := SystemTime,
                                 MessageType := MessageType.CMD,
                                 Severity    := Severity.DEBUG,
                                 MessageCode := 0,
                                 MessageText := 'SyncDefaultDynamics: Synchronization of DefaultDynamics triggered by RC, SyncMode = {1}, SyncTime = {2}, SyncDirection = PLC -> RC',
                                 Para1       :=  SYNC_MODE_TO_STRING(AxesGroup.Parameter.Plc.Parameter.SynchronizationModes.DefaultDynamics[SyncTime.AFTER_START_UP]),
                                 Para2       :=  SYNC_TIME_TO_STRING(SyncTime.AFTER_START_UP));
                                 RETURN;
			 END_IF
       
       // set timeout
       SetTimeout(PT := _rTimeout, rTimer := _rTimer);
       // jump back
      _rStep := 10;

       
  // ------------------------------------------
  // SyncMode : SERVER_TO_CLIENT 
  // ------------------------------------------
  12 : // Conflict triggerd by PLC ?  
       IF ( NOT AxesGroup.State.SyncStatePlc.InSync.DefaultDynamics )
       THEN
         // set timeout
         SetTimeout(PT := _rTimeout, rTimer := _rTimer);
         // inc step counter
        _rStep := 20; // -> read RC data and write it to PLC                  

         // Create log entry
         CreateLogMessagePara2 ( Timestamp   := SystemTime,
                                 MessageType := MessageType.CMD,
                                 Severity    := Severity.DEBUG,
                                 MessageCode := 0,
                                 MessageText := 'SyncDefaultDynamics: Synchronization of DefaultDynamics triggered by PLC, SyncMode = {1}, SyncTime = {2}, SyncDirection = RC -> PLC',
                                 Para1       :=  SYNC_MODE_TO_STRING(AxesGroup.Parameter.Plc.Parameter.SynchronizationModes.DefaultDynamics[SyncTime.AFTER_START_UP]),
                                 Para2       :=  SYNC_TIME_TO_STRING(SyncTime.AFTER_START_UP));
                                 RETURN;
       END_IF
   
       // Conflict triggered by RC ?
       IF ( NOT AxesGroup.State.SyncStateRc.InSync.DefaultDynamics )
       THEN
         // set timeout
         SetTimeout(PT := _rTimeout, rTimer := _rTimer);
         // inc step counter
        _rStep := 20; // -> read RC data and write it to PLC

         // Create log entry
         CreateLogMessagePara2 ( Timestamp   := SystemTime,
                                 MessageType := MessageType.CMD,
                                 Severity    := Severity.DEBUG,
                                 MessageCode := 0,
                                 MessageText := 'SyncDefaultDynamics: Synchronization of DefaultDynamics triggered by RC, SyncMode = {1}, SyncTime = {2}, SyncDirection = RC -> PLC',
                                 Para1       :=  SYNC_MODE_TO_STRING(AxesGroup.Parameter.Plc.Parameter.SynchronizationModes.DefaultDynamics[SyncTime.AFTER_START_UP]),
                                 Para2       :=  SYNC_TIME_TO_STRING(SyncTime.AFTER_START_UP));
                                 RETURN;
			 END_IF
       
       // set timeout
       SetTimeout(PT := _rTimeout, rTimer := _rTimer);
       // jump back
      _rStep := 10;
  

  // ------------------------------------------
  // SyncMode : AUTOMATIC 
  // ------------------------------------------
  13 : // Conflict triggerd by PLC ?  
       IF ( NOT AxesGroup.State.SyncStatePlc.InSync.DefaultDynamics )
       THEN
         // set timeout
         SetTimeout(PT := _rTimeout, rTimer := _rTimer);
         // inc step counter
        _rStep := 30; // -> write PLC data to RC                  
         
         // Create log entry
         CreateLogMessagePara2 ( Timestamp   := SystemTime,
                                 MessageType := MessageType.CMD,
                                 Severity    := Severity.DEBUG,
                                 MessageCode := 0,
                                 MessageText := 'SyncDefaultDynamics: Synchronization of DefaultDynamics triggered by PLC, SyncMode = {1}, SyncTime = {2}, SyncDirection = PLC -> RC',
                                 Para1       :=  SYNC_MODE_TO_STRING(AxesGroup.Parameter.Plc.Parameter.SynchronizationModes.DefaultDynamics[SyncTime.AFTER_START_UP]),
                                 Para2       :=  SYNC_TIME_TO_STRING(SyncTime.AFTER_START_UP));
                                 RETURN;
       END_IF
   
       // Conflict triggered by RC ?
       IF ( NOT AxesGroup.State.SyncStateRc.InSync.DefaultDynamics )
       THEN
         // set timeout
         SetTimeout(PT := _rTimeout, rTimer := _rTimer);
         // inc step counter
        _rStep := 20; // -> read RC data an write it to PLC

         // Create log entry
         CreateLogMessagePara2 ( Timestamp   := SystemTime,
                                 MessageType := MessageType.CMD,
                                 Severity    := Severity.DEBUG,
                                 MessageCode := 0,
                                 MessageText := 'SyncDefaultDynamics: Synchronization of DefaultDynamics triggered by RC, SyncMode = {1}, SyncTime = {2}, SyncDirection = RC -> PLC',
                                 Para1       :=  SYNC_MODE_TO_STRING(AxesGroup.Parameter.Plc.Parameter.SynchronizationModes.DefaultDynamics[SyncTime.AFTER_START_UP]),
                                 Para2       :=  SYNC_TIME_TO_STRING(SyncTime.AFTER_START_UP));
                                 RETURN;
			 END_IF
       
       // set timeout
       SetTimeout(PT := _rTimeout, rTimer := _rTimer);
       // jump back
      //_rStep := 10;


  // ------------------------------------------
  // Read Data from RC and write it to PLC
  // ------------------------------------------
  20 : IF (( NOT _readRobotDefaultDynamics.Busy  ) AND 
           ( NOT _readRobotDefaultDynamics.Error ))
       THEN
         // execute command
        _readRobotDefaultDynamics.Execute := TRUE;
         // set timeout
         SetTimeout(PT := _rTimeout, rTimer := _rTimer);
         // inc step counter
        _rStep := _rStep + 1;
       ELSE
         // check error ? 
         IF (_readRobotDefaultDynamics.Error)
         THEN
           ErrorID     := _readRobotDefaultDynamics.ErrorID;
           ErrorAddTxt := _readRobotDefaultDynamics.ErrorAddTxt;
         END_IF  
       
         // timeout exceeded ? 
         IF (CheckTimeout(_rTimer) = RobotLibraryConstants.OK)
         THEN
           ErrorID     := RobotLibraryErrorIdEnum.ERR_TIMEOUT_CMD;
           ErrorAddTxt := CONCAT(_stepName, DINT_TO_STRING(_rStep));
         END_IF
       END_IF
 
  21 : IF (( NOT _readRobotDefaultDynamics.Busy  ) AND
           ( NOT _readRobotDefaultDynamics.Error ) AND
           (     _readRobotDefaultDynamics.Done  ))
       THEN
         // reset execution
        _readRobotDefaultDynamics.Execute := FALSE;
         // update internal DefaultDynamics data
         DefaultDynamics := _readRobotDefaultDynamics.OutCmd.DynamicValues;         
        _defaultDynamics := _readRobotDefaultDynamics.OutCmd.DynamicValues;
         // set timeout
         SetTimeout(PT := _rTimeout, rTimer := _rTimer);
         // inc step counter
        _rStep := 10; // -> jump to after startup           
       ELSE
         // check error ? 
         IF (_readRobotDefaultDynamics.Error)
         THEN
           ErrorID     := _readRobotDefaultDynamics.ErrorID;
           ErrorAddTxt := _readRobotDefaultDynamics.ErrorAddTxt;           
         END_IF  
       
         // timeout exceeded ? 
         IF (CheckTimeout(_rTimer) = RobotLibraryConstants.OK)
         THEN
           ErrorID     := RobotLibraryErrorIdEnum.ERR_TIMEOUT_CMD;
           ErrorAddTxt := CONCAT(_stepName, DINT_TO_STRING(_rStep));
         END_IF
       END_IF


  // ------------------------------------------
  // Write data from PLC to RC
  // ------------------------------------------
  30 : IF (( NOT _writeRobotDefaultDynamics.Busy  ) AND 
           ( NOT _writeRobotDefaultDynamics.Error ))
       THEN
         // set command parameter
        _writeRobotDefaultDynamics.ParCmd.DynamicValues :=  DefaultDynamics;
         // execute command
        _writeRobotDefaultDynamics.Execute := TRUE;
         // set timeout
         SetTimeout(PT := _rTimeout, rTimer := _rTimer);
         // inc step counter
        _rStep := _rStep + 1;
       ELSE
         // check error ? 
         IF (_writeRobotDefaultDynamics.Error)
         THEN
           ErrorID     := _writeRobotDefaultDynamics.ErrorID;
           ErrorAddTxt := _writeRobotDefaultDynamics.ErrorAddTxt;;
         END_IF  
       
         // timeout exceeded ? 
         IF (CheckTimeout(_rTimer) = RobotLibraryConstants.OK)
         THEN
           ErrorID     := RobotLibraryErrorIdEnum.ERR_TIMEOUT_CMD;
           ErrorAddTxt := CONCAT(_stepName, DINT_TO_STRING(_rStep));
         END_IF
       END_IF
 
  31 : IF (( NOT _writeRobotDefaultDynamics.Busy  ) AND
           ( NOT _writeRobotDefaultDynamics.Error ) AND
           (     _writeRobotDefaultDynamics.Done  ))
       THEN
         // execute command
        _writeRobotDefaultDynamics.Execute := FALSE;      
         // update internal DefaultDynamics data
        _defaultDynamics := DefaultDynamics; 
         // set timeout
         SetTimeout(PT := _rTimeout, rTimer := _rTimer);
         // inc step counter
        _rStep := 10; // -> jump to after startup;           
       ELSE
         // check error ? 
         IF (_writeRobotDefaultDynamics.Error)
         THEN
           SetWarning( WarningID := RobotLibraryWarningIdEnum.WARN_DEFAULT_DYNAMICS_SYNC_FAILED_BY_ERROR_OF_READ_OR_WRITE_CMD, Overwrite := TRUE);    
         END_IF  
       
         // timeout exceeded ? 
         IF (CheckTimeout(_rTimer) = RobotLibraryConstants.OK)
         THEN
           ErrorID     := RobotLibraryErrorIdEnum.ERR_TIMEOUT_CMD;
           ErrorAddTxt := CONCAT(_stepName, DINT_TO_STRING(_rStep));
         END_IF
       END_IF
       
ELSE
  // invalid step
  ErrorID     := RobotLibraryErrorIdEnum.ERR_INVALID_STEP;
  ErrorAddTxt := CONCAT(_stepName , DINT_TO_STRING(_stepCmd));
END_CASE  
                
END_METHOD

METHOD PRIVATE HandleSyncRobotReferenceDynamics
VAR_IN_OUT
   /// Robot assignment of function
  AxesGroup         : AxesGroup;
  /// Reference dynamics stored on PLC. For more information refer to 5.5.7
  ReferenceDynamics : ReferenceDynamics;
END_VAR 

VAR
  /// Internal step counter name
 _stepName        : STRING;    
  /// Internal reference to step counter
 _rStep           : REFERENCE TO DINT;
  /// Internal reference to timer
 _rTimer          : REFERENCE TO TON;
  /// Internal reference to timeout
 _rTimeout        : REFERENCE TO TIME; 
  /// Internal reference to synchroniztion index
 _rSyncIdx        : REFERENCE TO USINT;
  /// internal bit for condition found
 _found           : BOOL;
  /// empty data set to reset all DataChanged bits
 _dataChangedNone : AxesGroupStateDataChanged;
END_VAR
                  // Set internal references 
_stepName      :=   '_stepSyncReferenceDynamics = ';
_rStep       REF=    _stepSyncReferenceDynamics;
_rTimer      REF=   _timerSyncReferenceDynamics;
_rTimeout    REF= _timeoutSyncReferenceDynamics;

CASE _rStep
OF    
  0: // Check initialisation configured ?
     IF (( _parCfg.PLC.Parameter.SynchronizationModes.ReferenceDynamics[SyncTime.DURING_START_UP] = SyncMode.NO_SYNCHRONIZATION ) AND
         ( _parCfg.PLC.Parameter.SynchronizationModes.ReferenceDynamics[SyncTime. AFTER_START_UP] = SyncMode.NO_SYNCHRONIZATION ))
     THEN
       RETURN;
     END_IF

     // wait for initialisation done
     IF  ((     AxesGroup.State.RobotData.RCSupportedFunctions .ReadRobotReferenceDynamics ) AND
          (     AxesGroup.State.RobotData.RCSupportedFunctions.WriteRobotReferenceDynamics ) AND
          (     AxesGroup.State.Initialized                                              ) AND 
          ( NOT Error                                                                    ))  
     THEN
       // Create log entry
       CreateLogMessagePara1 ( Timestamp   := SystemTime,
                               MessageType := MessageType.CMD,
                               Severity    := Severity.DEBUG,
                               MessageCode := 0,
                               MessageText := 'SyncReferenceDynamics: Start initial reading of ReferenceDynamics from RC',
                               Para1       :=  '');
       
       // set timeout
       SetTimeout(PT := _rTimeout, rTimer := _rTimer);
       // inc step counter
      _rStep := _rStep + 1;
     END_IF     

     
     // Start read ReferenceDynamics
  1: IF (( NOT _readRobotReferenceDynamics.Busy  ) AND 
         ( NOT _readRobotReferenceDynamics.Error ) AND
         ( NOT _readRobotReferenceDynamics.Done  ))
     THEN
       // execute command
      _readRobotReferenceDynamics.Execute := TRUE;
       // set timeout
       SetTimeout(PT := _rTimeout, rTimer := _rTimer);
       // inc step counter
      _rStep := _rStep + 1;
     ELSE
       // check error ? 
       IF ( _readRobotReferenceDynamics.Error )
       THEN
         SetWarning( WarningID := RobotLibraryWarningIdEnum.WARN_REFERENCE_DYNAMICS_SYNC_FAILED_BY_ERROR_OF_READ_OR_WRITE_CMD, Overwrite := FALSE);           
       END_IF  
       
       // timeout exceeded ? 
       IF (CheckTimeout(_rTimer) = RobotLibraryConstants.OK)
       THEN
         ErrorID     := RobotLibraryErrorIdEnum.ERR_TIMEOUT_CMD;
         ErrorAddTxt := CONCAT(_stepName, DINT_TO_STRING(_rStep));
       END_IF
     END_IF
 
     
     // Wait ReferenceDynamics read
  2: IF (( NOT _readRobotReferenceDynamics.Busy  ) AND
         ( NOT _readRobotReferenceDynamics.Error ) AND
         (     _readRobotReferenceDynamics.Done  ))
     THEN
       // reset execution
      _readRobotReferenceDynamics.Execute := FALSE;
       // Copy data
      _referenceDynamics := _readRobotReferenceDynamics.OutCmd.DynamicValues;
       // Set plc in sync flag
       AxesGroup.State.SyncStatePlc.InSync.ReferenceDynamics := TRUE;
       // inc step counter
      _rStep := _rStep + 1;           

       // Check ReferenceDynamics data is equal ? 
       IF ( NOT IsReferenceDynamicsEqual( Data1 := _referenceDynamics, Data2 := ReferenceDynamics, IgnoreTimestamp := TRUE))
       THEN
         // Reset plc in sync flag
         AxesGroup.State.SyncStatePlc.InSync.ReferenceDynamics := FALSE;
         // Set data changed flag
         AxesGroup.State.DataChanged.ReferenceDynamics := TRUE;
         // set timeout
         SetTimeout(PT := _rTimeout, rTimer := _rTimer);
        
         // Create log entry
         CreateLogMessagePara1 ( Timestamp   := SystemTime,
                                 MessageType := MessageType.CMD,
                                 Severity    := Severity.DEBUG,
                                 MessageCode := 0,
                                 MessageText := 'SyncReferenceDynamics: Detected a difference in ReferenceDynamics between PLC and RC',
                                 Para1       :=  '');
        
        
         // Check synchronisation is enabled ? 
         IF ( NOT  AxesGroup.State.DataEnableSync.EnableSyncReferenceDynamics )
         THEN
           SetInfo ( InfoID := RobotLibraryInfoIdEnum.INFO_SYNC_REFERENCE_DYNAMICS_DISABLED, Overwrite := FALSE );
				 END_IF
         
         // Check user interaction needed ?  
         IF ( AxesGroup.Parameter.Plc.Parameter.SyncUserInteraction.ReferenceDynamics )
         THEN
           SetWarning ( WarningID := RobotLibraryWarningIdEnum.WARN_REFERENCE_DYNAMICS_SYNC_ERROR, Overwrite := FALSE );                    
				 END_IF
			 END_IF             
     ELSE
       // check error ? 
       IF (_readRobotReferenceDynamics.Error)
       THEN
         // Set warning
         SetWarning( WarningID := RobotLibraryWarningIdEnum.WARN_REFERENCE_DYNAMICS_SYNC_FAILED_BY_ERROR_OF_READ_OR_WRITE_CMD, Overwrite := TRUE);                    
       END_IF  
       
       // timeout exceeded ? 
       IF (CheckTimeout(_rTimer) = RobotLibraryConstants.OK)
       THEN
         ErrorID     := RobotLibraryErrorIdEnum.ERR_TIMEOUT_CMD;
         ErrorAddTxt := CONCAT(_stepName, DINT_TO_STRING(_rStep));
       END_IF
     END_IF
     
     
     // Check synchronisation state ? 
  3: IF ((  NOT AxesGroup.State.DataChanged.ReferenceDynamics                                                                                    ) OR 
         (      AxesGroup.Parameter.Plc.Parameter.SynchronizationModes.ReferenceDynamics[SyncTime.DURING_START_UP] = SyncMode.NO_SYNCHRONIZATION ))
     THEN
       // Update bit for data in sync
       AxesGroup.State.SyncStatePlc.InSync.ReferenceDynamics := NOT AxesGroup.State.DataChanged.ReferenceDynamics ;
       // set timeout
       SetTimeout(PT := _rTimeout, rTimer := _rTimer);
       // inc step counter
      _rStep := 10; // -> jump to after startup
            
       // Create log entry
       CreateLogMessagePara1 ( Timestamp   := SystemTime,
                               MessageType := MessageType.CMD,
                               Severity    := Severity.DEBUG,
                               MessageCode := 0,
                               MessageText := 'SyncReferenceDynamics: Synchronization Startup Phase done',
                               Para1       :=  '' );      
     ELSE 
       // Check user interaction needed ? 
       IF ( NOT AxesGroup.Parameter.Plc.Parameter.SyncUserInteraction.ReferenceDynamics )
       THEN 
         CASE AxesGroup.Parameter.Plc.Parameter.SynchronizationModes.ReferenceDynamics[SyncTime.DURING_START_UP] OF

           SyncMode.SERVER_TO_CLIENT : 

             // Overwrite PLC data with RC data
             ReferenceDynamics := _referenceDynamics;            
             // Reset data changed flags
             AxesGroup.State.DataChanged.ReferenceDynamics := _dataChangedNone.ReferenceDynamics;
             // Reset Synchronizing flag
             AxesGroup.State.Synchronizing.ReferenceDynamics := FALSE;
             // Set plc in sync flag
             AxesGroup.State.SyncStatePlc.InSync.ReferenceDynamics := TRUE;
             // set timeout
             SetTimeout(PT := _rTimeout, rTimer := _rTimer);
             // inc step counter
            _rStep := 10; // -> jump to after startup         

            // Create log entry
            CreateLogMessagePara2 ( Timestamp   := SystemTime,
                                    MessageType := MessageType.CMD,
                                    Severity    := Severity.DEBUG,
                                    MessageCode := 0,
                                    MessageText := 'SyncReferenceDynamics: Synchronization of ReferenceDynamics triggered by StartUp-Compare, SyncMode = {1}, SyncTime = {2}, SyncDirection = RC -> PLC',
                                    Para1       :=  SYNC_MODE_TO_STRING(AxesGroup.Parameter.Plc.Parameter.SynchronizationModes.ReferenceDynamics[SyncTime.DURING_START_UP]),
                                    Para2       :=  SYNC_TIME_TO_STRING(SyncTime.DURING_START_UP));
            // Create log entry
            CreateLogMessagePara1 ( Timestamp   := SystemTime,
                                    MessageType := MessageType.CMD,
                                    Severity    := Severity.DEBUG,
                                    MessageCode := 0,
                                    MessageText := 'SyncReferenceDynamics: Applied the initial read ReferenceDynamics from RC',
                                    Para1       :=  '' );

				   SyncMode.CLIENT_TO_SERVER : ;

             IF ( AxesGroup.State.DataChanged.ReferenceDynamics ) 
             THEN
               // Reset plc in sync flag
               AxesGroup.State.SyncStatePlc.InSync.ReferenceDynamics := FALSE;
               // Set Synchronizing flag
               AxesGroup.State.Synchronizing.ReferenceDynamics := TRUE;
               // set timeout
               SetTimeout(PT := _rTimeout, rTimer := _rTimer);
               // inc step counter
              _rStep := _rStep +1; // -> write PLC data to RC                  
               // Create log entry
               CreateLogMessagePara2 ( Timestamp   := SystemTime,
                                       MessageType := MessageType.CMD,
                                       Severity    := Severity.DEBUG,
                                       MessageCode := 0,
                                       MessageText := 'SyncReferenceDynamics: Synchronization of ReferenceDynamics triggered by StartUp-Compare, SyncMode = {1}, SyncTime = {2}, SyncDirection = PLC -> RC',
                                       Para1       :=  SYNC_MODE_TO_STRING(AxesGroup.Parameter.Plc.Parameter.SynchronizationModes.ReferenceDynamics[SyncTime.DURING_START_UP]),
                                       Para2       :=  SYNC_TIME_TO_STRING(SyncTime.DURING_START_UP));
             ELSE
               // Reset data changed flags
               AxesGroup.State.DataChanged.ReferenceDynamics := _dataChangedNone.ReferenceDynamics;
               // Reset Synchronizing flag
               AxesGroup.State.Synchronizing.ReferenceDynamics := FALSE;
               // Set plc in sync flag
               AxesGroup.State.SyncStatePlc.InSync.ReferenceDynamics := TRUE;
               // set timeout
               SetTimeout(PT := _rTimeout, rTimer := _rTimer);
               // inc step counter
              _rStep := 10; // -> jump to after startup                  
				     END_IF
         ELSE
           // invalid sync mode for startup
           SetError( ErrorID := RobotLibraryErrorIdEnum.ERR_SYNC_MODE_INVALID, Overwrite := TRUE );
 	       END_CASE
       END_IF
     END_IF  

     
     // Start write ReferenceDynamics data  
  4: IF (( NOT _writeRobotReferenceDynamics.Busy  ) AND 
         ( NOT _writeRobotReferenceDynamics.Error ))
     THEN
       // set command parameter
      _writeRobotReferenceDynamics.ParCmd.DynamicValues :=  ReferenceDynamics;
       // execute command
      _writeRobotReferenceDynamics.Execute := TRUE;
       // set timeout
       SetTimeout(PT := _rTimeout, rTimer := _rTimer);
       // inc step counter
      _rStep := _rStep + 1;
     ELSE
       // check error ? 
       IF (_writeRobotReferenceDynamics.Error)
       THEN
         ErrorID     := _writeRobotReferenceDynamics.ErrorID;
         ErrorAddTxt := _writeRobotReferenceDynamics.ErrorAddTxt;;
       END_IF  
       
       // timeout exceeded ? 
       IF (CheckTimeout(_rTimer) = RobotLibraryConstants.OK)
       THEN
         ErrorID     := RobotLibraryErrorIdEnum.ERR_TIMEOUT_CMD;
         ErrorAddTxt := CONCAT(_stepName, DINT_TO_STRING(_rStep));
       END_IF
     END_IF
 
     
     // Wait ReferenceDynamics data written ?   
  5: IF (( NOT _writeRobotReferenceDynamics.Busy  ) AND
         ( NOT _writeRobotReferenceDynamics.Error ) AND
         (     _writeRobotReferenceDynamics.Done  ))
     THEN
       // execute command
      _writeRobotReferenceDynamics.Execute := FALSE;
       // apply ReferenceDynamics data to internal ReferenceDynamics data
      _referenceDynamics := ReferenceDynamics;
       // reset data changed bit 
       AxesGroup.State.DataChanged.ReferenceDynamics := FALSE;
       // set timeout        
       SetTimeout(PT := _rTimeout, rTimer := _rTimer);
       // dec step counter
      _rStep := _rStep - 2; 
     ELSE
       // check error ? 
       IF (_writeRobotReferenceDynamics.Error)
       THEN
         SetWarning( WarningID := RobotLibraryWarningIdEnum.WARN_REFERENCE_DYNAMICS_SYNC_FAILED_BY_ERROR_OF_READ_OR_WRITE_CMD, Overwrite := TRUE);           
       END_IF  
       
       // timeout exceeded ? 
       IF (CheckTimeout(_rTimer) = RobotLibraryConstants.OK)
       THEN
         ErrorID     := RobotLibraryErrorIdEnum.ERR_TIMEOUT_CMD;
         ErrorAddTxt := CONCAT(_stepName, DINT_TO_STRING(_rStep));
       END_IF
     END_IF

     
  // --------------------------------------------
  // SyncMode after startup : 
  // --------------------------------------------
         
  10 : // check synchronisation active ? 
       IF ( AxesGroup.Parameter.Plc.Parameter.SynchronizationModes.ReferenceDynamics[SyncTime.AFTER_START_UP] = SyncMode.NO_SYNCHRONIZATION)
       THEN
         RETURN;
       END_IF

       // compare ReferenceDynamics data
       AxesGroup.State.DataChanged.ReferenceDynamics := NOT IsReferenceDynamicsEqual( Data1 := ReferenceDynamics, Data2 := _referenceDynamics, IgnoreTimestamp := FALSE);

       // Check ReferenceDynamics data changed ? 
       IF (AxesGroup.State.DataChanged.ReferenceDynamics)
       THEN
         // Create log entry
         CreateLogMessagePara1 ( Timestamp   := SystemTime,
                                 MessageType := MessageType.CMD,
                                 Severity    := Severity.DEBUG,
                                 MessageCode := 0,
                                 MessageText := 'SyncReferenceDynamics: Detected a local change of ReferenceDynamics on PLC, SyncTime = {1}',
                                 Para1       :=  SYNC_TIME_TO_STRING(SyncTime.AFTER_START_UP));       
       END_IF

       // Update plc in sync flag
       AxesGroup.State.SyncStatePlc.InSync.ReferenceDynamics := NOT AxesGroup.State.DataChanged.ReferenceDynamics; 


       // Check synchronization is needed ? 
       IF ( NOT AxesGroup.State.SyncStatePlc.InSync.ReferenceDynamics ) XOR  
          ( NOT AxesGroup.State.SyncStateRc .InSync.ReferenceDynamics )
       THEN
         CASE AxesGroup.Parameter.Plc.Parameter.SynchronizationModes.ReferenceDynamics[SyncTime.AFTER_START_UP] 
         OF         
           // NO_SYNCHRONIZATION
           SyncMode.NO_SYNCHRONIZATION : ; // no further action 
           
           // CLIENT_TO_SERVER
           SyncMode.CLIENT_TO_SERVER :
             // set timeout
             SetTimeout(PT := _rTimeout, rTimer := _rTimer);
             // inc step counter
            _rStep := 11;
  
           // SERVER_TO_CLIENT
           SyncMode.SERVER_TO_CLIENT :
             // set timeout
             SetTimeout(PT := _rTimeout, rTimer := _rTimer);
             // inc step counter
            _rStep := 12;
  
           // AUTOMATIC
           SyncMode.AUTOMATIC : 
             // set timeout
             SetTimeout(PT := _rTimeout, rTimer := _rTimer);
             // inc step counter
            _rStep := 13;
         END_CASE
       ELSE
         // datas changeḍ on both sides ? -> Warning 
         IF (( NOT AxesGroup.State.SyncStatePlc.InSync.ReferenceDynamics ) AND  
             ( NOT AxesGroup.State.SyncStateRc .InSync.ReferenceDynamics ))
         THEN
           SetWarning( WarningID := RobotLibraryWarningIdEnum.WARN_REFERENCE_DYNAMICS_SYNC_BOTH_SIDES_CHANGED, Overwrite := TRUE);
         END_IF
       END_IF


  // ------------------------------------------
  // SyncMode : CLIENT_TO_SERVER 
  // ------------------------------------------  
  11 : // Conflict triggerd by PLC ?  
       IF ( NOT AxesGroup.State.SyncStatePlc.InSync.ReferenceDynamics ) 
       THEN
         // set timeout
         SetTimeout(PT := _rTimeout, rTimer := _rTimer);
         // inc step counter
        _rStep := 30; // -> write PLC data to RC                  
         
         // Create log entry
         CreateLogMessagePara2 ( Timestamp   := SystemTime,
                                 MessageType := MessageType.CMD,
                                 Severity    := Severity.DEBUG,
                                 MessageCode := 0,
                                 MessageText := 'SyncReferenceDynamics: Synchronization of ReferenceDynamics triggered by PLC, SyncMode = {1}, SyncTime = {2}, SyncDirection = PLC -> RC',
                                 Para1       :=  SYNC_MODE_TO_STRING(AxesGroup.Parameter.Plc.Parameter.SynchronizationModes.ReferenceDynamics[SyncTime.AFTER_START_UP]),
                                 Para2       :=  SYNC_TIME_TO_STRING(SyncTime.AFTER_START_UP));
                                 RETURN;
       END_IF
   
       // Conflict triggered by RC ?
       IF ( NOT AxesGroup.State.SyncStateRc.InSync.ReferenceDynamics )
       THEN
         // set timeout
         SetTimeout(PT := _rTimeout, rTimer := _rTimer);
         // inc step counter
        _rStep := 30; // -> write PLC data to RC

         // Create log entry
         CreateLogMessagePara2 ( Timestamp   := SystemTime,
                                 MessageType := MessageType.CMD,
                                 Severity    := Severity.DEBUG,
                                 MessageCode := 0,
                                 MessageText := 'SyncReferenceDynamics: Synchronization of ReferenceDynamics triggered by RC, SyncMode = {1}, SyncTime = {2}, SyncDirection = PLC -> RC',
                                 Para1       :=  SYNC_MODE_TO_STRING(AxesGroup.Parameter.Plc.Parameter.SynchronizationModes.ReferenceDynamics[SyncTime.AFTER_START_UP]),
                                 Para2       :=  SYNC_TIME_TO_STRING(SyncTime.AFTER_START_UP));
                                 RETURN;
			 END_IF
       
       // set timeout
       SetTimeout(PT := _rTimeout, rTimer := _rTimer);
       // jump back
      _rStep := 10;

       
  // ------------------------------------------
  // SyncMode : SERVER_TO_CLIENT 
  // ------------------------------------------
  12 : // Conflict triggerd by PLC ?  
       IF ( NOT AxesGroup.State.SyncStatePlc.InSync.ReferenceDynamics )
       THEN
         // set timeout
         SetTimeout(PT := _rTimeout, rTimer := _rTimer);
         // inc step counter
        _rStep := 20; // -> read RC data and write it to PLC                  

         // Create log entry
         CreateLogMessagePara2 ( Timestamp   := SystemTime,
                                 MessageType := MessageType.CMD,
                                 Severity    := Severity.DEBUG,
                                 MessageCode := 0,
                                 MessageText := 'SyncReferenceDynamics: Synchronization of ReferenceDynamics triggered by PLC, SyncMode = {1}, SyncTime = {2}, SyncDirection = RC -> PLC',
                                 Para1       :=  SYNC_MODE_TO_STRING(AxesGroup.Parameter.Plc.Parameter.SynchronizationModes.ReferenceDynamics[SyncTime.AFTER_START_UP]),
                                 Para2       :=  SYNC_TIME_TO_STRING(SyncTime.AFTER_START_UP));
                                 RETURN;
       END_IF
   
       // Conflict triggered by RC ?
       IF ( NOT AxesGroup.State.SyncStateRc.InSync.ReferenceDynamics )
       THEN
         // set timeout
         SetTimeout(PT := _rTimeout, rTimer := _rTimer);
         // inc step counter
        _rStep := 20; // -> read RC data and write it to PLC

         // Create log entry
         CreateLogMessagePara2 ( Timestamp   := SystemTime,
                                 MessageType := MessageType.CMD,
                                 Severity    := Severity.DEBUG,
                                 MessageCode := 0,
                                 MessageText := 'SyncReferenceDynamics: Synchronization of ReferenceDynamics triggered by RC, SyncMode = {1}, SyncTime = {2}, SyncDirection = RC -> PLC',
                                 Para1       :=  SYNC_MODE_TO_STRING(AxesGroup.Parameter.Plc.Parameter.SynchronizationModes.ReferenceDynamics[SyncTime.AFTER_START_UP]),
                                 Para2       :=  SYNC_TIME_TO_STRING(SyncTime.AFTER_START_UP));
                                 RETURN;
			 END_IF
       
       // set timeout
       SetTimeout(PT := _rTimeout, rTimer := _rTimer);
       // jump back
      _rStep := 10;
  

  // ------------------------------------------
  // SyncMode : AUTOMATIC 
  // ------------------------------------------
  13 : // Conflict triggerd by PLC ?  
       IF ( NOT AxesGroup.State.SyncStatePlc.InSync.ReferenceDynamics )
       THEN
         // set timeout
         SetTimeout(PT := _rTimeout, rTimer := _rTimer);
         // inc step counter
        _rStep := 30; // -> write PLC data to RC                  
         
         // Create log entry
         CreateLogMessagePara2 ( Timestamp   := SystemTime,
                                 MessageType := MessageType.CMD,
                                 Severity    := Severity.DEBUG,
                                 MessageCode := 0,
                                 MessageText := 'SyncReferenceDynamics: Synchronization of ReferenceDynamics triggered by PLC, SyncMode = {1}, SyncTime = {2}, SyncDirection = PLC -> RC',
                                 Para1       :=  SYNC_MODE_TO_STRING(AxesGroup.Parameter.Plc.Parameter.SynchronizationModes.ReferenceDynamics[SyncTime.AFTER_START_UP]),
                                 Para2       :=  SYNC_TIME_TO_STRING(SyncTime.AFTER_START_UP));
                                 RETURN;
       END_IF
   
       // Conflict triggered by RC ?
       IF ( NOT AxesGroup.State.SyncStateRc.InSync.ReferenceDynamics )
       THEN
         // set timeout
         SetTimeout(PT := _rTimeout, rTimer := _rTimer);
         // inc step counter
        _rStep := 20; // -> read RC data an write it to PLC

         // Create log entry
         CreateLogMessagePara2 ( Timestamp   := SystemTime,
                                 MessageType := MessageType.CMD,
                                 Severity    := Severity.DEBUG,
                                 MessageCode := 0,
                                 MessageText := 'SyncReferenceDynamics: Synchronization of ReferenceDynamics triggered by RC, SyncMode = {1}, SyncTime = {2}, SyncDirection = RC -> PLC',
                                 Para1       :=  SYNC_MODE_TO_STRING(AxesGroup.Parameter.Plc.Parameter.SynchronizationModes.ReferenceDynamics[SyncTime.AFTER_START_UP]),
                                 Para2       :=  SYNC_TIME_TO_STRING(SyncTime.AFTER_START_UP));
                                 RETURN;
			 END_IF
       
       // set timeout
       SetTimeout(PT := _rTimeout, rTimer := _rTimer);
       // jump back
      //_rStep := 10;


  // ------------------------------------------
  // Read Data from RC and write it to PLC
  // ------------------------------------------
  20 : IF (( NOT _readRobotReferenceDynamics.Busy  ) AND 
           ( NOT _readRobotReferenceDynamics.Error ))
       THEN
         // execute command
        _readRobotReferenceDynamics.Execute := TRUE;
         // set timeout
         SetTimeout(PT := _rTimeout, rTimer := _rTimer);
         // inc step counter
        _rStep := _rStep + 1;
       ELSE
         // check error ? 
         IF (_readRobotReferenceDynamics.Error)
         THEN
           ErrorID     := _readRobotReferenceDynamics.ErrorID;
           ErrorAddTxt := _readRobotReferenceDynamics.ErrorAddTxt;
         END_IF  
       
         // timeout exceeded ? 
         IF (CheckTimeout(_rTimer) = RobotLibraryConstants.OK)
         THEN
           ErrorID     := RobotLibraryErrorIdEnum.ERR_TIMEOUT_CMD;
           ErrorAddTxt := CONCAT(_stepName, DINT_TO_STRING(_rStep));
         END_IF
       END_IF
 
  21 : IF (( NOT _readRobotReferenceDynamics.Busy  ) AND
           ( NOT _readRobotReferenceDynamics.Error ) AND
           (     _readRobotReferenceDynamics.Done  ))
       THEN
         // reset execution
        _readRobotReferenceDynamics.Execute := FALSE;
         // update internal ReferenceDynamics data
         ReferenceDynamics := _readRobotReferenceDynamics.OutCmd.DynamicValues;         
        _referenceDynamics := _readRobotReferenceDynamics.OutCmd.DynamicValues;
         // set timeout
         SetTimeout(PT := _rTimeout, rTimer := _rTimer);
         // inc step counter
        _rStep := 10; // -> jump to after startup           
       ELSE
         // check error ? 
         IF (_readRobotReferenceDynamics.Error)
         THEN
           ErrorID     := _readRobotReferenceDynamics.ErrorID;
           ErrorAddTxt := _readRobotReferenceDynamics.ErrorAddTxt;           
         END_IF  
       
         // timeout exceeded ? 
         IF (CheckTimeout(_rTimer) = RobotLibraryConstants.OK)
         THEN
           ErrorID     := RobotLibraryErrorIdEnum.ERR_TIMEOUT_CMD;
           ErrorAddTxt := CONCAT(_stepName, DINT_TO_STRING(_rStep));
         END_IF
       END_IF


